ACTION Correction:
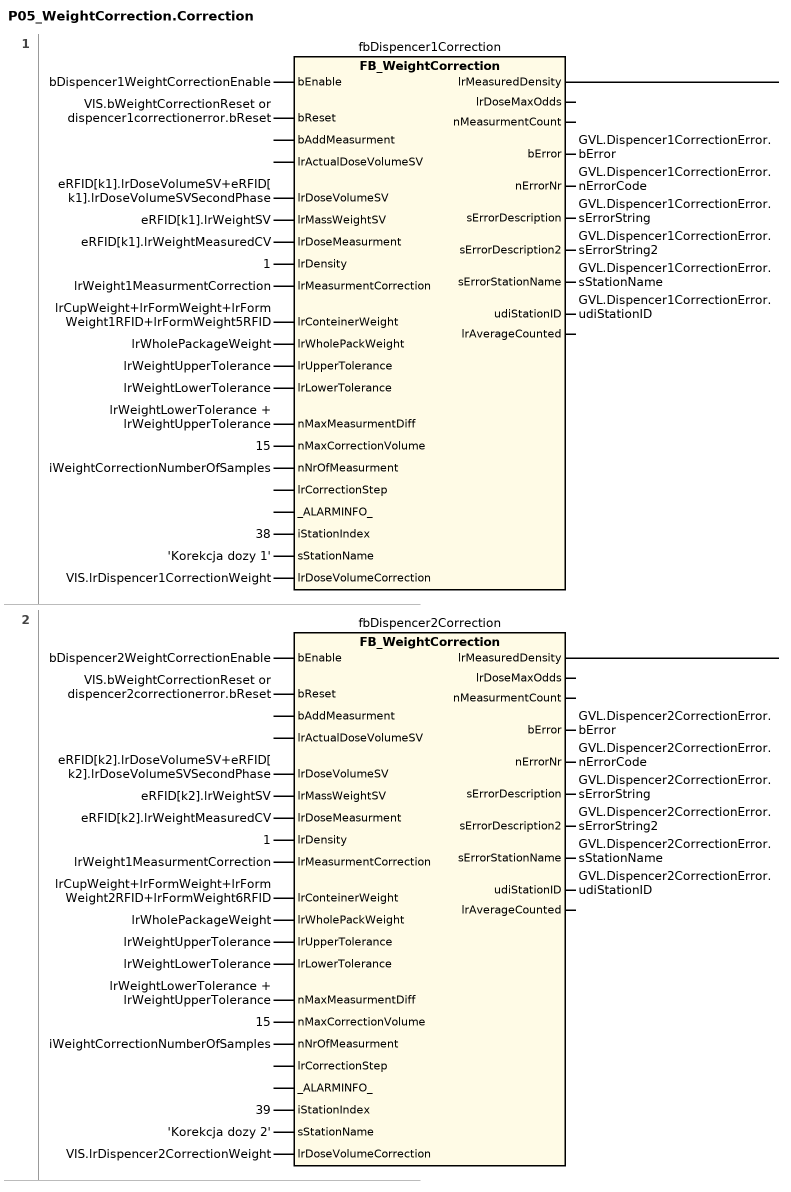
// NETWORK 1
fbDispencer1Correction(
    bEnable := bDispencer1WeightCorrectionEnable,
    bReset := VIS.bWeightCorrectionReset or dispencer1correctionerror.bReset,
    lrDoseVolumeSV := eRFID[k1].lrDoseVolumeSV+eRFID[k1].lrDoseVolumeSVSecondPhase,
    lrMassWeightSV := eRFID[k1].lrWeightSV,
    lrDoseMeasurment := eRFID[k1].lrWeightMeasuredCV,
    lrDensity := 1,
    lrMeasurmentCorrection := lrWeight1MeasurmentCorrection,
    lrConteinerWeight := lrCupWeight+lrFormWeight+lrFormWeight1RFID+lrFormWeight5RFID,
    lrWholePackWeight := lrWholePackageWeight,
    lrUpperTolerance := lrWeightUpperTolerance,
    lrLowerTolerance := lrWeightLowerTolerance,
    nMaxMeasurmentDiff := lrWeightLowerTolerance + lrWeightUpperTolerance,
    nMaxCorrectionVolume := 15,
    nNrOfMeasurment := iWeightCorrectionNumberOfSamples,
    iStationIndex := 38,
    sStationName := 'Korekcja dozy 1',
    lrDoseVolumeCorrection := VIS.lrDispencer1CorrectionWeight,
    bError => GVL.Dispencer1CorrectionError.bError,
    nErrorNr => GVL.Dispencer1CorrectionError.nErrorCode,
    sErrorDescription => GVL.Dispencer1CorrectionError.sErrorString,
    sErrorDescription2 => GVL.Dispencer1CorrectionError.sErrorString2,
    sErrorStationName => GVL.Dispencer1CorrectionError.sStationName,
    udiStationID => GVL.Dispencer1CorrectionError.udiStationID); // FB_WeightCorrection

// NETWORK 2
fbDispencer2Correction(
    bEnable := bDispencer2WeightCorrectionEnable,
    bReset := VIS.bWeightCorrectionReset or dispencer2correctionerror.bReset,
    lrDoseVolumeSV := eRFID[k2].lrDoseVolumeSV+eRFID[k2].lrDoseVolumeSVSecondPhase,
    lrMassWeightSV := eRFID[k2].lrWeightSV,
    lrDoseMeasurment := eRFID[k2].lrWeightMeasuredCV,
    lrDensity := 1,
    lrMeasurmentCorrection := lrWeight1MeasurmentCorrection,
    lrConteinerWeight := lrCupWeight+lrFormWeight+lrFormWeight2RFID+lrFormWeight6RFID,
    lrWholePackWeight := lrWholePackageWeight,
    lrUpperTolerance := lrWeightUpperTolerance,
    lrLowerTolerance := lrWeightLowerTolerance,
    nMaxMeasurmentDiff := lrWeightLowerTolerance + lrWeightUpperTolerance,
    nMaxCorrectionVolume := 15,
    nNrOfMeasurment := iWeightCorrectionNumberOfSamples,
    iStationIndex := 39,
    sStationName := 'Korekcja dozy 2',
    lrDoseVolumeCorrection := VIS.lrDispencer2CorrectionWeight,
    bError => GVL.Dispencer2CorrectionError.bError,
    nErrorNr => GVL.Dispencer2CorrectionError.nErrorCode,
    sErrorDescription => GVL.Dispencer2CorrectionError.sErrorString,
    sErrorDescription2 => GVL.Dispencer2CorrectionError.sErrorString2,
    sErrorStationName => GVL.Dispencer2CorrectionError.sStationName,
    udiStationID => GVL.Dispencer2CorrectionError.udiStationID); // FB_WeightCorrection

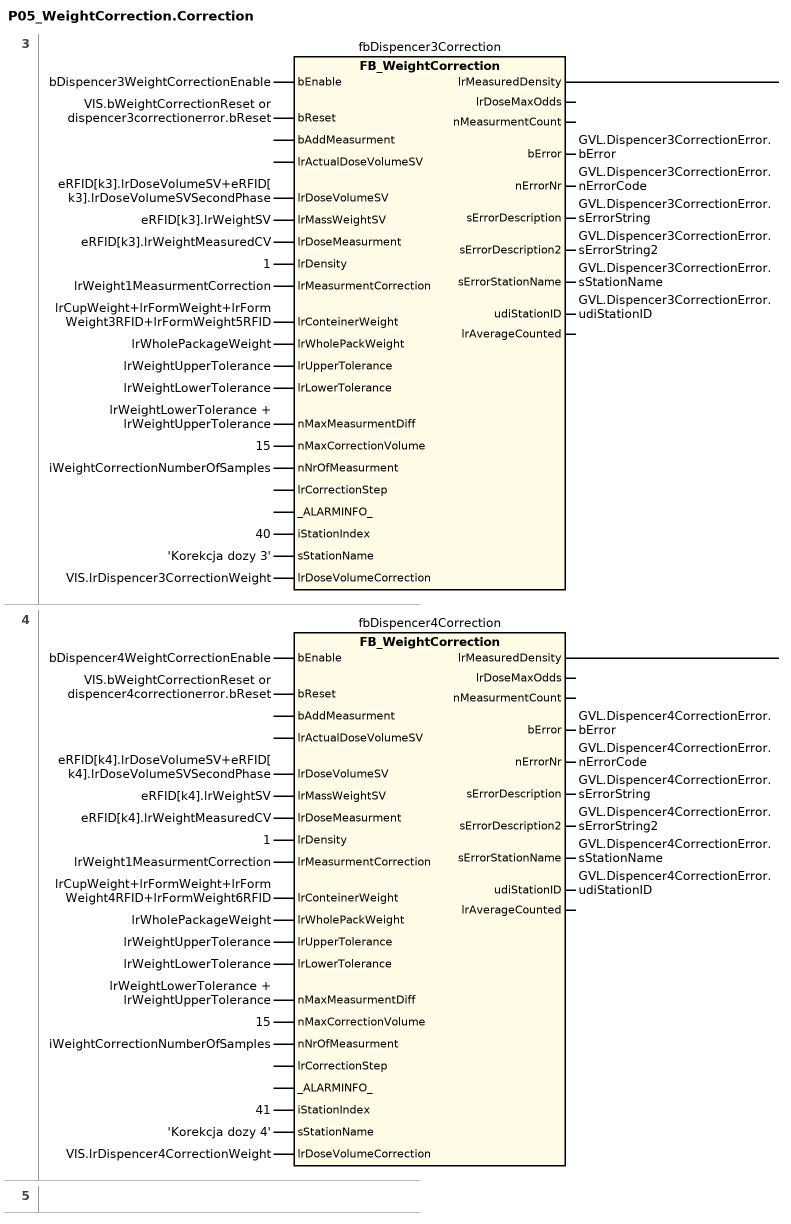
// NETWORK 3
fbDispencer3Correction(
    bEnable := bDispencer3WeightCorrectionEnable,
    bReset := VIS.bWeightCorrectionReset or dispencer3correctionerror.bReset,
    lrDoseVolumeSV := eRFID[k3].lrDoseVolumeSV+eRFID[k3].lrDoseVolumeSVSecondPhase,
    lrMassWeightSV := eRFID[k3].lrWeightSV,
    lrDoseMeasurment := eRFID[k3].lrWeightMeasuredCV,
    lrDensity := 1,
    lrMeasurmentCorrection := lrWeight1MeasurmentCorrection,
    lrConteinerWeight := lrCupWeight+lrFormWeight+lrFormWeight3RFID+lrFormWeight5RFID,
    lrWholePackWeight := lrWholePackageWeight,
    lrUpperTolerance := lrWeightUpperTolerance,
    lrLowerTolerance := lrWeightLowerTolerance,
    nMaxMeasurmentDiff := lrWeightLowerTolerance + lrWeightUpperTolerance,
    nMaxCorrectionVolume := 15,
    nNrOfMeasurment := iWeightCorrectionNumberOfSamples,
    iStationIndex := 40,
    sStationName := 'Korekcja dozy 3',
    lrDoseVolumeCorrection := VIS.lrDispencer3CorrectionWeight,
    bError => GVL.Dispencer3CorrectionError.bError,
    nErrorNr => GVL.Dispencer3CorrectionError.nErrorCode,
    sErrorDescription => GVL.Dispencer3CorrectionError.sErrorString,
    sErrorDescription2 => GVL.Dispencer3CorrectionError.sErrorString2,
    sErrorStationName => GVL.Dispencer3CorrectionError.sStationName,
    udiStationID => GVL.Dispencer3CorrectionError.udiStationID); // FB_WeightCorrection

// NETWORK 4
fbDispencer4Correction(
    bEnable := bDispencer4WeightCorrectionEnable,
    bReset := VIS.bWeightCorrectionReset or dispencer4correctionerror.bReset,
    lrDoseVolumeSV := eRFID[k4].lrDoseVolumeSV+eRFID[k4].lrDoseVolumeSVSecondPhase,
    lrMassWeightSV := eRFID[k4].lrWeightSV,
    lrDoseMeasurment := eRFID[k4].lrWeightMeasuredCV,
    lrDensity := 1,
    lrMeasurmentCorrection := lrWeight1MeasurmentCorrection,
    lrConteinerWeight := lrCupWeight+lrFormWeight+lrFormWeight4RFID+lrFormWeight6RFID,
    lrWholePackWeight := lrWholePackageWeight,
    lrUpperTolerance := lrWeightUpperTolerance,
    lrLowerTolerance := lrWeightLowerTolerance,
    nMaxMeasurmentDiff := lrWeightLowerTolerance + lrWeightUpperTolerance,
    nMaxCorrectionVolume := 15,
    nNrOfMeasurment := iWeightCorrectionNumberOfSamples,
    iStationIndex := 41,
    sStationName := 'Korekcja dozy 4',
    lrDoseVolumeCorrection := VIS.lrDispencer4CorrectionWeight,
    bError => GVL.Dispencer4CorrectionError.bError,
    nErrorNr => GVL.Dispencer4CorrectionError.nErrorCode,
    sErrorDescription => GVL.Dispencer4CorrectionError.sErrorString,
    sErrorDescription2 => GVL.Dispencer4CorrectionError.sErrorString2,
    sErrorStationName => GVL.Dispencer4CorrectionError.sStationName,
    udiStationID => GVL.Dispencer4CorrectionError.udiStationID); // FB_WeightCorrection

// NETWORK 5
END_ACTION

ACTION OnePhaseDosing:
	(*******Dozowanie jednofazowe*****)

IF rtWeightingDone.Q THEN //Triger, wszystko wazy się jednoczesnie
	
	FOR i := 1 TO 100 DO
		
		IF  eWeightPackageState[1].nCardNumber = eRFID[i].nCardNumber AND eRFID[i].nDispencerNr=1 THEN	 
			
			fbDispencer1Correction.bAddMeasurment:=(eRFID[i].nDispencerNr=1 AND bDispencer1WeightCorrectionEnable) AND 
								(eRFID[i].lrDoseVolumeCV>(0.5*eRFID[i].lrDoseVolumeSV) OR eRFID[i].lrDoseVolumeCVSecondPhase>(0.5*eRFID[i].lrDoseVolumeSVSecondPhase)) AND
								(eRFID[i].lrWeightMeasuredCV>0);															
			k1:=i;	//Zapamiętywanie numeru tablicy		
			
			IF 					(eRFID[i].nDispencerNr=1 AND bDispencer1WeightCorrectionEnable) AND 
								((eRFID[i].lrDoseVolumeCV>(0.5*eRFID[i].lrDoseVolumeSV)) OR (eRFID[i].lrDoseVolumeCVSecondPhase>(0.5*eRFID[i].lrDoseVolumeSVSecondPhase))) AND
								(eRFID[i].lrWeightMeasuredCV>0) THEN
				iCorectTest:=iCorectTest+1;	
			END_IF;	
		END_IF	
    
		IF  eWeightPackageState[1].nCardNumber = eRFID[i].nCardNumber AND eRFID[i].nDispencerNr=2 THEN	
 
			fbDispencer2Correction.bAddMeasurment := (eRFID[i].nDispencerNr=2 AND bDispencer2WeightCorrectionEnable) AND 
								(eRFID[i].lrDoseVolumeCV>(0.5*eRFID[i].lrDoseVolumeSV) OR eRFID[i].lrDoseVolumeCVSecondPhase>(0.5*eRFID[i].lrDoseVolumeSVSecondPhase)) AND 
								(eRFID[i].lrWeightMeasuredCV>0);
			k2:=i;	//Zapamiętywanie numeru tablicy	
			iCorectTest2:=iCorectTest2+1;							
		END_IF
		
		IF  eWeightPackageState[1].nCardNumber = eRFID[i].nCardNumber AND eRFID[i].nDispencerNr=3 THEN	 
			fbDispencer3Correction.bAddMeasurment := (eRFID[i].nDispencerNr=3 AND bDispencer3WeightCorrectionEnable) AND 
								(eRFID[i].lrDoseVolumeCV>(0.5*eRFID[i].lrDoseVolumeSV) OR eRFID[i].lrDoseVolumeCVSecondPhase>(0.5*eRFID[i].lrDoseVolumeSVSecondPhase)) AND 
								(eRFID[i].lrWeightMeasuredCV>0);						
			k3:=i;	//Zapamiętywanie numeru tablicy		
			iCorectTest3:=iCorectTest3+1;					
		END_IF	
		
		IF  eWeightPackageState[1].nCardNumber = eRFID[i].nCardNumber AND eRFID[i].nDispencerNr=4 THEN	 
			fbDispencer4Correction.bAddMeasurment := (eRFID[i].nDispencerNr=4 AND bDispencer4WeightCorrectionEnable) AND 
								(eRFID[i].lrDoseVolumeCV>(0.5*eRFID[i].lrDoseVolumeSV) OR eRFID[i].lrDoseVolumeCVSecondPhase>(0.5*eRFID[i].lrDoseVolumeSVSecondPhase)) AND 
								(eRFID[i].lrWeightMeasuredCV>0);					
			k4:=i;	//Zapamiętywanie numeru tablicy	
			iCorectTest4:=iCorectTest4+1;						
		END_IF
		
	END_FOR
	
	
	FOR i := 1 TO 100 DO
		
		IF  eWeightPackageState[2].nCardNumber = eRFID[i].nCardNumber AND eRFID[i].nDispencerNr=1 THEN	 
			fbDispencer1Correction.bAddMeasurment:=(eRFID[i].nDispencerNr=1 AND bDispencer1WeightCorrectionEnable) AND 
								(eRFID[i].lrDoseVolumeCV>(0.5*eRFID[i].lrDoseVolumeSV) OR eRFID[i].lrDoseVolumeCVSecondPhase>(0.5*eRFID[i].lrDoseVolumeSVSecondPhase)) AND
								(eRFID[i].lrWeightMeasuredCV>0);															
			k1:=i;	//Zapamiętywanie numeru tablicy						
		END_IF	
		
		IF  eWeightPackageState[2].nCardNumber = eRFID[i].nCardNumber AND eRFID[i].nDispencerNr=2 THEN	 
			fbDispencer2Correction.bAddMeasurment := (eRFID[i].nDispencerNr=2 AND bDispencer2WeightCorrectionEnable) AND 
								(eRFID[i].lrDoseVolumeCV>(0.5*eRFID[i].lrDoseVolumeSV) OR eRFID[i].lrDoseVolumeCVSecondPhase>(0.5*eRFID[i].lrDoseVolumeSVSecondPhase)) AND 
								(eRFID[i].lrWeightMeasuredCV>0);
			k2:=i;	//Zapamiętywanie numeru tablicy						
		END_IF
		
		IF  eWeightPackageState[2].nCardNumber = eRFID[i].nCardNumber AND eRFID[i].nDispencerNr=3 THEN	 
			fbDispencer3Correction.bAddMeasurment := (eRFID[i].nDispencerNr=3 AND bDispencer3WeightCorrectionEnable) AND 
								(eRFID[i].lrDoseVolumeCV>(0.5*eRFID[i].lrDoseVolumeSV) OR eRFID[i].lrDoseVolumeCVSecondPhase>(0.5*eRFID[i].lrDoseVolumeSVSecondPhase)) AND 
								(eRFID[i].lrWeightMeasuredCV>0);						
			k3:=i;	//Zapamiętywanie numeru tablicy						
		END_IF	
		
		IF  eWeightPackageState[2].nCardNumber = eRFID[i].nCardNumber AND eRFID[i].nDispencerNr=4 THEN	 
			fbDispencer4Correction.bAddMeasurment := (eRFID[i].nDispencerNr=4 AND bDispencer4WeightCorrectionEnable) AND 
								(eRFID[i].lrDoseVolumeCV>(0.5*eRFID[i].lrDoseVolumeSV) OR eRFID[i].lrDoseVolumeCVSecondPhase>(0.5*eRFID[i].lrDoseVolumeSVSecondPhase)) AND 
								(eRFID[i].lrWeightMeasuredCV>0);					
			k4:=i;	//Zapamiętywanie numeru tablicy						
		END_IF
		
	END_FOR		
    
	FOR i := 1 TO 100 DO
		
		IF  eWeightPackageState[3].nCardNumber = eRFID[i].nCardNumber  AND eRFID[i].nDispencerNr=1 THEN	 
			fbDispencer1Correction.bAddMeasurment:=(eRFID[i].nDispencerNr=1 AND bDispencer1WeightCorrectionEnable) AND 
								(eRFID[i].lrDoseVolumeCV>(0.5*eRFID[i].lrDoseVolumeSV) OR eRFID[i].lrDoseVolumeCVSecondPhase>(0.5*eRFID[i].lrDoseVolumeSVSecondPhase)) AND
								(eRFID[i].lrWeightMeasuredCV>0);															
			k1:=i;	//Zapamiętywanie numeru tablicy						
		END_IF	
		
		IF  eWeightPackageState[3].nCardNumber = eRFID[i].nCardNumber AND eRFID[i].nDispencerNr=2 THEN	 
			fbDispencer2Correction.bAddMeasurment := (eRFID[i].nDispencerNr=2 AND bDispencer2WeightCorrectionEnable) AND 
								(eRFID[i].lrDoseVolumeCV>(0.5*eRFID[i].lrDoseVolumeSV) OR eRFID[i].lrDoseVolumeCVSecondPhase>(0.5*eRFID[i].lrDoseVolumeSVSecondPhase)) AND 
								(eRFID[i].lrWeightMeasuredCV>0);
			k2:=i;	//Zapamiętywanie numeru tablicy						
		END_IF
		
		IF  eWeightPackageState[3].nCardNumber = eRFID[i].nCardNumber AND eRFID[i].nDispencerNr=3 THEN	 
			fbDispencer3Correction.bAddMeasurment := (eRFID[i].nDispencerNr=3 AND bDispencer3WeightCorrectionEnable) AND 
								(eRFID[i].lrDoseVolumeCV>(0.5*eRFID[i].lrDoseVolumeSV) OR eRFID[i].lrDoseVolumeCVSecondPhase>(0.5*eRFID[i].lrDoseVolumeSVSecondPhase)) AND 
								(eRFID[i].lrWeightMeasuredCV>0);						
			k3:=i;	//Zapamiętywanie numeru tablicy						
		END_IF	
		
		IF  eWeightPackageState[3].nCardNumber = eRFID[i].nCardNumber AND eRFID[i].nDispencerNr=4 THEN	 
			fbDispencer4Correction.bAddMeasurment := (eRFID[i].nDispencerNr=4 AND bDispencer4WeightCorrectionEnable) AND 
								(eRFID[i].lrDoseVolumeCV>(0.5*eRFID[i].lrDoseVolumeSV) OR eRFID[i].lrDoseVolumeCVSecondPhase>(0.5*eRFID[i].lrDoseVolumeSVSecondPhase)) AND 
								(eRFID[i].lrWeightMeasuredCV>0);					
			k4:=i;	//Zapamiętywanie numeru tablicy						
		END_IF
		
	END_FOR
    
	FOR i := 1 TO 100 DO
		
		IF  eWeightPackageState[4].nCardNumber = eRFID[i].nCardNumber AND eRFID[i].nDispencerNr=1 THEN	 
			fbDispencer1Correction.bAddMeasurment:=(eRFID[i].nDispencerNr=1 AND bDispencer1WeightCorrectionEnable) AND 
								(eRFID[i].lrDoseVolumeCV>(0.5*eRFID[i].lrDoseVolumeSV) OR eRFID[i].lrDoseVolumeCVSecondPhase>(0.5*eRFID[i].lrDoseVolumeSVSecondPhase)) AND
								(eRFID[i].lrWeightMeasuredCV>0);															
			k1:=i;	//Zapamiętywanie numeru tablicy						
		END_IF	
		
		IF  eWeightPackageState[4].nCardNumber = eRFID[i].nCardNumber AND eRFID[i].nDispencerNr=2 THEN	 
			fbDispencer2Correction.bAddMeasurment := (eRFID[i].nDispencerNr=2 AND bDispencer2WeightCorrectionEnable) AND 
								(eRFID[i].lrDoseVolumeCV>(0.5*eRFID[i].lrDoseVolumeSV) OR eRFID[i].lrDoseVolumeCVSecondPhase>(0.5*eRFID[i].lrDoseVolumeSVSecondPhase)) AND 
								(eRFID[i].lrWeightMeasuredCV>0);
			k2:=i;	//Zapamiętywanie numeru tablicy						
		END_IF
		
		IF  eWeightPackageState[4].nCardNumber = eRFID[i].nCardNumber AND eRFID[i].nDispencerNr=3 THEN	 
			fbDispencer3Correction.bAddMeasurment := (eRFID[i].nDispencerNr=3 AND bDispencer3WeightCorrectionEnable) AND 
								(eRFID[i].lrDoseVolumeCV>(0.5*eRFID[i].lrDoseVolumeSV) OR eRFID[i].lrDoseVolumeCVSecondPhase>(0.5*eRFID[i].lrDoseVolumeSVSecondPhase)) AND 
								(eRFID[i].lrWeightMeasuredCV>0);						
			k3:=i;	//Zapamiętywanie numeru tablicy						
		END_IF
	
		IF  eWeightPackageState[4].nCardNumber = eRFID[i].nCardNumber AND eRFID[i].nDispencerNr=4 THEN	 
			fbDispencer4Correction.bAddMeasurment := (eRFID[i].nDispencerNr=4 AND bDispencer4WeightCorrectionEnable) AND 
								(eRFID[i].lrDoseVolumeCV>(0.5*eRFID[i].lrDoseVolumeSV) OR eRFID[i].lrDoseVolumeCVSecondPhase>(0.5*eRFID[i].lrDoseVolumeSVSecondPhase)) AND 
								(eRFID[i].lrWeightMeasuredCV>0);					
			k4:=i;	//Zapamiętywanie numeru tablicy						
		END_IF
		
	END_FOR

END_IF
END_ACTION

ACTION TwoPhaseDosing:
	(*******Dozowanie jednofazowe*****)

IF rtWeightingDone.Q THEN //Triger, wszystko wazy się jednoczesnie
	
	FOR i2 := 1 TO 100 DO
		
		IF  eWeightPackage2PhasePackageState[1].nCardNumber = eRFID[i2].nCardNumber AND (*eRFID[i2].nDispencerNr=1*) eRFID[i2].nDispencerNrSecondPhase=1 THEN	 
			
			fbDispencer1Correction.bAddMeasurment:=((*eRFID[i2].nDispencerNr=1 AND*) eRFID[i2].nDispencerNrSecondPhase=1 AND bDispencer1WeightCorrectionEnable) AND 
								(eRFID[i2].lrDoseVolumeCV>(0.5*eRFID[i2].lrDoseVolumeSV) OR eRFID[i2].lrDoseVolumeCVSecondPhase>(0.5*eRFID[i2].lrDoseVolumeSVSecondPhase)) AND
								(eRFID[i2].lrWeightMeasuredCV>0);															
			k1:=i2;	//Zapamiętywanie numeru tablicy		
			iCorectTest:=iCorectTest+1;
		END_IF	
	END_FOR
	
	FOR i3:=1 TO 100 DO
	
    (*
		IF  eWeightPackage2PhasePackageState[1].nCardNumber = eRFID[i2].nCardNumber AND (*eRFID[i2].nDispencerNr=2*) eRFID[i2].nDispencerNrSecondPhase=2 THEN	
 
			fbDispencer2Correction.bAddMeasurment := ((*eRFID[i2].nDispencerNr=2*)eRFID[i2].nDispencerNrSecondPhase=2 AND bDispencer2WeightCorrectionEnable) AND 
								(eRFID[i2].lrDoseVolumeCV>(0.5*eRFID[i2].lrDoseVolumeSV) OR eRFID[i2].lrDoseVolumeCVSecondPhase>(0.5*eRFID[i2].lrDoseVolumeSVSecondPhase)) AND 
								(eRFID[i2].lrWeightMeasuredCV>0);
			k2:=i2;	//Zapamiętywanie numeru tablicy	
			iCorectTest2:=iCorectTest2+1;	
			EXIT;						
		END_IF
	*)	
		IF  eWeightPackage2PhasePackageState[1].nCardNumber = eRFID[i3].nCardNumber AND eRFID[i3].nDispencerNr=3 THEN	 
			fbDispencer3Correction.bAddMeasurment := (eRFID[i3].nDispencerNr=3 AND bDispencer3WeightCorrectionEnable) AND 
								(eRFID[i3].lrDoseVolumeCV>(0.5*eRFID[i3].lrDoseVolumeSV) OR eRFID[i3].lrDoseVolumeCVSecondPhase>(0.5*eRFID[i3].lrDoseVolumeSVSecondPhase)) AND 
								(eRFID[i3].lrWeightMeasuredCV>0);						
			k3:=i3;	//Zapamiętywanie numeru tablicy		
			iCorectTest3:=iCorectTest3+1;	
						
		END_IF	
	(*	
		IF  eWeightPackage2PhasePackageState[1].nCardNumber = eRFID[i2].nCardNumber AND eRFID[i2].nDispencerNr=4 THEN	 
			fbDispencer4Correction.bAddMeasurment := (eRFID[i2].nDispencerNr=4 AND bDispencer4WeightCorrectionEnable) AND 
								(eRFID[i2].lrDoseVolumeCV>(0.5*eRFID[i2].lrDoseVolumeSV) OR eRFID[i2].lrDoseVolumeCVSecondPhase>(0.5*eRFID[i2].lrDoseVolumeSVSecondPhase)) AND 
								(eRFID[i2].lrWeightMeasuredCV>0);					
			k4:=i2;	//Zapamiętywanie numeru tablicy	
			iCorectTest4:=iCorectTest4+1;	
			EXIT;					
		END_IF
	*)	

	END_FOR
	
	
	FOR i4 := 1 TO 100 DO
		(*
		IF  eWeightPackage2PhasePackageState[2].nCardNumber = eRFID[i].nCardNumber AND eRFID[i].nDispencerNr=1 THEN	 
			fbDispencer1Correction.bAddMeasurment:=(eRFID[i].nDispencerNr=1 AND bDispencer1WeightCorrectionEnable) AND 
								(eRFID[i].lrDoseVolumeCV>(0.5*eRFID[i].lrDoseVolumeSV) OR eRFID[i].lrDoseVolumeCVSecondPhase>(0.5*eRFID[i].lrDoseVolumeSVSecondPhase)) AND
								(eRFID[i].lrWeightMeasuredCV>0);															
			k1:=i;	//Zapamiętywanie numeru tablicy	
			iCorectTest5:=iCorectTest5+1;	
		EXIT;			
		END_IF	
		*)
		IF  eWeightPackage2PhasePackageState[2].nCardNumber = eRFID[i4].nCardNumber AND (*eRFID[i].nDispencerNr=2*) eRFID[i4].nDispencerNrSecondPhase=2 THEN	 
			fbDispencer2Correction.bAddMeasurment := ((*eRFID[i].nDispencerNr=2*) eRFID[i4].nDispencerNrSecondPhase=2 AND bDispencer2WeightCorrectionEnable) AND 
								(eRFID[i4].lrDoseVolumeCV>(0.5*eRFID[i4].lrDoseVolumeSV) OR eRFID[i4].lrDoseVolumeCVSecondPhase>(0.5*eRFID[i4].lrDoseVolumeSVSecondPhase)) AND 
								(eRFID[i4].lrWeightMeasuredCV>0);
			k2:=i4;	//Zapamiętywanie numeru tablicy		
			iCorectTest6:=iCorectTest6+1;	
		END_IF
	END_FOR
	
	FOR i5:=1 TO 100 DO
		(*
		IF  eWeightPackage2PhasePackageState[2].nCardNumber = eRFID[i].nCardNumber AND eRFID[i].nDispencerNr=3 THEN	 
			fbDispencer3Correction.bAddMeasurment := (eRFID[i].nDispencerNr=3 AND bDispencer3WeightCorrectionEnable) AND 
								(eRFID[i].lrDoseVolumeCV>(0.5*eRFID[i].lrDoseVolumeSV) OR eRFID[i].lrDoseVolumeCVSecondPhase>(0.5*eRFID[i].lrDoseVolumeSVSecondPhase)) AND 
								(eRFID[i].lrWeightMeasuredCV>0);						
			k3:=i;	//Zapamiętywanie numeru tablicy	
			iCorectTest7:=iCorectTest7+1;	
		EXIT	;			
		END_IF	
		*)
		IF  eWeightPackage2PhasePackageState[2].nCardNumber = eRFID[i5].nCardNumber AND eRFID[i5].nDispencerNr=4  THEN	 
			fbDispencer4Correction.bAddMeasurment := (eRFID[i5].nDispencerNr=4 AND bDispencer4WeightCorrectionEnable) AND 
								(eRFID[i5].lrDoseVolumeCV>(0.5*eRFID[i5].lrDoseVolumeSV) OR eRFID[i5].lrDoseVolumeCVSecondPhase>(0.5*eRFID[i5].lrDoseVolumeSVSecondPhase)) AND 
								(eRFID[i5].lrWeightMeasuredCV>0);					
			k4:=i5;	//Zapamiętywanie numeru tablicy	
			iCorectTest8:=iCorectTest8+1;	
		END_IF
		
	END_FOR		
    


END_IF
END_ACTION

END_PROGRAM

// ---- POUs/FB/FB_WeightCorrection.TcPOU
(*
Nazwa:			FB_WeightCorrection
Opis:			Korekcja wagi
Wersja:			v1.3
Data:			2019-11-28
Autor:			TW,DP
Urzadzenia:		Korekta wagi 
Konfiguracja:	
Info: 
-wyłączono wpisywanie maksymalnej korekty bo to bez sensu, ze wpisywało np -15
-poprawiono warningi, które wskazywalo w kompilatorze
-poprawiony blad maksymalnej korekty (minus przerabia na plus)
*)

FUNCTION_BLOCK FB_WeightCorrection
VAR_INPUT
	bEnable:BOOL;					//Zezwolenie na pracę automatycznej korekcji
	bReset:BOOL;					//Reset korekcji dozy i obliczonej gęstości
	bAddMeasurment:BOOL;			//Dodanie pomiaru wagi do rozpatrzenia korekcji dozy
	lrActualDoseVolumeSV:LREAL;		//Aktualna wartość nastawy objetości dozy (ta która jest nastawiona na dozowniku)
	lrDoseVolumeSV:LREAL;			//Wartość nastawy objetości dozy dla danego opakowania (wartość z rejestru)  [ml]
	lrMassWeightSV:LREAL;			//Zadana wartość masy produktu [g]
	lrDoseMeasurment:LREAL;			//Wartość masy odczytana z wagi [g]
	lrDensity:LREAL;				//Gęstość masy g/ml (Jeśli wartość 0, oblicz z wydozowanej ostatniej wartości)
	lrMeasurmentCorrection:LREAL;	//Korekcja wskazania wagi [g]
	lrConteinerWeight:LREAL;			//Waga kubeczka [g]
	lrWholePackWeight:LREAL;		//Waga kubeczka razem z platynką i nakrętką itp. [g]
	lrUpperTolerance:LREAL;			//Górna granica tolerancji
	lrLowerTolerance:LREAL;			//Dolna granica tolerancji	
	nMaxMeasurmentDiff:LREAL;		//Maksymalna różnica pomiędzy pomiarami
	nMaxCorrectionVolume:UDINT;		//Maksymalna nastawa dozy korekcji
	nNrOfMeasurment:UINT;			//Ilość próbek do uśrednienia wartości korekcji dozy
	lrCorrectionStep: LREAL;		//Skok korekcji dozy [ml]
	_ALARMINFO_ :BOOL;
	iStationIndex:UDINT;					//Numer stacji 
	sStationName:STRING;					//Nazwa stacji	

END_VAR
VAR_OUTPUT
	lrMeasuredDensity:LREAL;		//Obliczona wartość gęstości [g/ml]
	lrDoseMaxOdds:LREAL;			//Najwieksze różnice pomiędzy wagami wydozowań
	nMeasurmentCount:UINT;			//Ilość zebranych pomiarów do uśrednienia wagi
	bError:BOOL; 					//Błąd korekcji <=0
	nErrorNr:UDINT;					//Numer Błędu
	sErrorDescription:STRING;		//Opis błędu 
	sErrorDescription2: STRING;				//Opis błędu 2
	sErrorStationName:STRING;				//Nazwa stacji
	udiStationID:UDINT;				// Nr stacji

	lrAverageCounted:LREAL;			//średnia z ostatnich pomiarów
END_VAR
VAR_IN_OUT
	lrDoseVolumeCorrection:LREAL;			//Wartość korekty dozy [ml]
END_VAR
VAR
	rtAddMeasurment: R_TRIG;
	aMeasuredWeight: ARRAY [1..10] OF LREAL;
	
	i: UINT;
	// Suma pomiarów wag
	lrMeasureSum: LREAL;
	// Średnia pomiarów wagi
	lrAverageWeight: LREAL;
	lrUsedDensity:LREAL;
	// trigger Resetu
	rtrigReset: R_TRIG;
	// poprzednia wartość dozy kontrolowanej butelki [ml]
	lrLastDoseVolumeSV: LREAL :=89033008911;
	lrDoseVolumeCorrectionTemp: LREAL;
	Delta: DINT;
	bWeightTooLow:BOOL;
	bWeightTooHigh:BOOL;
	lrWeightHisteresisCenter:LREAL;//
END_VAR

aStationID();
rtAddMeasurment(CLK:=bAddMeasurment,Q=>);


IF bEnable THEN
	
	
	//Jeśli odczytana nowa doza 
	IF rtAddMeasurment.Q THEN
		
		//Jeśli dozy różne zacznij próbkowanie wag od początku
		IF lrActualDoseVolumeSV<>lrDoseVolumeSV THEN
			nMeasurmentCount:=0;
			lrMeasureSum:=0;
		
		//jeśli nastawy zgadzają sie 	
		ELSE	
		
			lrLastDoseVolumeSV:=lrDoseVolumeSV;
			bError:=FALSE;
			nMeasurmentCount:=nMeasurmentCount+1;
			aMeasuredWeight[nMeasurmentCount]:=lrDoseMeasurment-lrConteinerWeight+lrMeasurmentCorrection;
			lrMeasureSum:=lrMeasureSum+aMeasuredWeight[nMeasurmentCount];
			
			IF nMeasurmentCount=1 THEN
				lrDoseMaxOdds:=0;
			END_IF
			
			//Sprawdzanie największych odchyłek w wadze miedzy pomiarami
			FOR i:=1 TO nMeasurmentCount DO
				IF ABS(aMeasuredWeight[i]-aMeasuredWeight[nMeasurmentCount])>lrDoseMaxOdds THEN
					lrDoseMaxOdds:=ABS(aMeasuredWeight[i]-aMeasuredWeight[nMeasurmentCount]);
				END_IF
			END_FOR
			

		END_IF
		
		IF lrDoseMaxOdds>nMaxMeasurmentDiff THEN
				nMeasurmentCount:=0;
				lrMeasureSum:=0;
		END_IF
		//Obliczanie korekty jeśli ilość próbek pomiarowych została osiągnięta
		IF nMeasurmentCount>=(nNrOfMeasurment) THEN
			lrAverageWeight:=lrMeasureSum/UINT_TO_LREAL(nMeasurmentCount);
			lrAverageCounted:=lrAverageWeight;
			lrMeasureSum:=0;
			//lrMeasuredDensity:=(lrAverageWeight)/(lrDoseVolumeSV(*+lrDoseVolumeCorrection*)+0.000000000001);
			IF lrDensity>0 THEN
				lrUsedDensity:=lrDensity;
			ELSE
				//lrUsedDensity:=lrMeasuredDensity;
				bError:=TRUE;
				nErrorNr:=211;
				sErrorDescription:='Zadana wartość gęstości poniżej 0.';
			END_IF
			
			
			//Jeśli nie ma błędu oblicz korektę
			IF NOT bError (*AND (((LREAL_TO_DINT(lrMassWeightSV)-LREAL_TO_DINT(lrAverageWeight))>=ABS(lrLowerTolerance)) OR (((LREAL_TO_DINT(lrAverageWeight)-LREAL_TO_DINT(lrMassWeightSV)>=ABS(lrUpperTolerance)))))*) THEN
				
			
				Delta:=(LREAL_TO_DINT(lrMassWeightSV)-LREAL_TO_DINT(lrAverageCounted));
				
			//	lrWeightHisteresisCenter:=(LREAL_TO_DINT(lrMassWeightSV)+((ABS(lrLowerTolerance)+ABS(lrUpperTolerance))/2)-(ABS(lrLowerTolerance)));
				// 04.11.2022 Dązy do zadanej bez środka
				lrWeightHisteresisCenter:=lrMassWeightSV;
				
				//Wykrywanie czy waga przekracza górny zakres widełek
				IF LREAL_TO_DINT(lrAverageCounted)<LREAL_TO_DINT(lrWeightHisteresisCenter) THEN
					bWeightTooLow:=TRUE;
					bWeightTooHigh:=FALSE;
			   //Wykrywanie czy waga przekracza dolną granicę widełek
				ELSIF LREAL_TO_DINT(lrAverageCounted)>LREAL_TO_DINT(lrWeightHisteresisCenter)THEN
					bWeightTooLow:=FALSE;
					bWeightTooHigh:=TRUE;
				END_IF
				
				
				
				//Jeśli osiągnieta wartość miedzy widełkami wyłącz podnoszenie dozy
				IF LREAL_TO_DINT(lrAverageCounted)>=(LREAL_TO_DINT(lrMassWeightSV)+((ABS(lrLowerTolerance)+ABS(lrUpperTolerance))/2)-(ABS(lrLowerTolerance))) THEN
					bWeightTooLow:=FALSE;
				END_IF
				
				//Jeśli osiągnieta wartość miedzy widełkami wyłącz obniżanie dozy
				IF LREAL_TO_DINT(lrAverageCounted)<=(LREAL_TO_DINT(lrMassWeightSV)+((ABS(lrLowerTolerance)+ABS(lrUpperTolerance))/2)-(ABS(lrLowerTolerance)))THEN
					bWeightTooHigh:=FALSE;
				END_IF
				
				//Zwiększ dozę jeśli za mała wartość
				IF bWeightTooLow THEN
					IF ABS(LREAL_TO_DINT(lrMassWeightSV)-LREAL_TO_DINT(lrAverageCounted))>10 THEN
						;//lrDoseVolumeCorrection:=lrDoseVolumeCorrection+ABS(LREAL_TO_DINT(lrMassWeightSV)-LREAL_TO_DINT(lrAverageCounted));//wyłączone max
					ELSE
						lrDoseVolumeCorrection:=lrDoseVolumeCorrection+lrCorrectionStep;	
					END_IF
						
						lrLastDoseVolumeSV:=lrDoseVolumeSV;
						
				//Zmniejsz dozę jeśli za duża	
				ELSIF bWeightTooHigh THEN
					IF ABS(LREAL_TO_DINT(lrMassWeightSV)-LREAL_TO_DINT(lrAverageCounted))>10 THEN
						;//lrDoseVolumeCorrection:=lrDoseVolumeCorrection-ABS(LREAL_TO_DINT(lrMassWeightSV)-LREAL_TO_DINT(lrAverageCounted));
					ELSE
						lrDoseVolumeCorrection:=lrDoseVolumeCorrection-lrCorrectionStep;	
					END_IF
					
					lrLastDoseVolumeSV:=lrDoseVolumeSV;
				END_IF
				
				//jeśli korekta poza maksymalnym zakresem, przepisz maksymalny zakres
				IF lrDoseVolumeCorrection>nMaxCorrectionVolume THEN					
					lrDoseVolumeCorrection:=nMaxCorrectionVolume;	
				END_IF
				IF lrDoseVolumeCorrection<-UDINT_TO_LREAL(nMaxCorrectionVolume) THEN					
					lrDoseVolumeCorrection:=-UDINT_TO_LREAL(nMaxCorrectionVolume);	
				END_IF
				
			END_IF;
			nMeasurmentCount:=0;
			lrAverageWeight:=0;
		END_IF	
	END_IF

ELSE
	nMeasurmentCount:=0;
	bError:=FALSE;
	lrDoseMaxOdds:=0;
END_IF

rtrigReset(CLK:=bReset,Q=>);

IF rtrigReset.Q (*AND NOT bError *)THEN
	nMeasurmentCount:=0;
	bError:=FALSE;
	lrDoseMaxOdds:=0;
	lrDoseVolumeCorrection:=0;
	lrMeasuredDensity:=0;
	lrMeasureSum:=0;
END_IF

ErrorHandling();

ACTION aStationID:
udiStationID	:=	iStationIndex;
END_ACTION

ACTION ErrorHandling:

IF bReset THEN
	bError:=FALSE;
	nErrorNr:=0;
	sErrorDescription:='';
	lrDoseMaxOdds:=0;
	lrDoseVolumeCorrectionTemp:=0;
END_IF

IF bEnable THEN
	;
	
ELSE
	bError:=FALSE;
	nErrorNr:=0;
	sErrorDescription:='';	
END_IF


(*Przepisywanie nazwy stacji*)
sErrorStationName := sStationName;
END_ACTION

END_FUNCTION_BLOCK

// ---- POUs/Recipes/P010_AlarmsWarningsInfosLogs.TcPOU
PROGRAM P010_AlarmsWarningsInfosLogs
VAR CONSTANT 
	iNumberOfStations									:	DINT:=46;	
	iMaxNumberOfErrors									:	DINT:=100;	
	iStartLinePositionY									:	INT:=0;		
	iLinePositionYStep									:	INT:=55;
	iNumberOfWarnings									:	INT:=13;
END_VAR

VAR	
	bWarning				:	BOOL;	
	bHistoryShowScreeen		:BOOL;
	//Wiska
	udiInfoCounter			:	UDINT;
	sInfoBitmapId			:	STRING	:=	'MainImages.InfoOff'	;
	udiInfoTxtColor 		:	UDINT	:=	16#FFFFFFFF;

	udiWarningCounter		:	UDINT;
	sWarningBitmapId		:	STRING	:=	'MainImages.WarningOff'	;
	udiWarningTxtColor 		:	UDINT	:=	16#FFFFFFFF;


	iAlarmCounter			:	DINT;
	sAlarmBitmapId			:	STRING	:=	'MainImages.ErrorOff'	;
	udiAlarmTxtColor 		:	UDINT	:=	16#FFFFFFFF;
	//

	aiLinePositionYErrors										:	ARRAY [0..iNumberOfStations] OF INT;
	iLinePositionXErrors										:	INT	:=	50;
	iStationInErrorCounter											:	INT;					
	
	aiLinePositionYWarnings										:	ARRAY [0..iNumberOfWarnings - 1] OF INT;
	iLinePositionXWarnings										:	INT	:=	50;
	iStationInWarningCounter									:	INT;
	iPrevStationInWarningCounter								:	INT:=-1;
				
	//stError												: 	ARRAY[0..iMaxNumberOfErrors] OF ST_Error;
	aActualErrorsArray									:	ARRAY[0..2,0..iMaxNumberOfErrors] OF WSTRING(120);//iNumberOfWarnings - 1
	//stWarning											: 	ARRAY[0..iNumberOfWarnings - 1] OF ST_Warning;
	aActualWarningsArray								:	ARRAY[0..1,0..19] OF WSTRING(120);//iNumberOfWarnings - 1
	
	i													:	DINT;
	k													:	INT;
	j													:	INT;
	
	diId												:	DINT	:=	-1;
	iPrevStationInErrorCounter							:	DINT	:=	-1;

	udiResetCase										:	UDINT;
	artReset											:	ARRAY [0..iMaxNumberOfErrors] OF R_TRIG;
	abReset												:	ARRAY [0.. iMaxNumberOfErrors] OF BOOL;
	udiWarningResetCase									:	UDINT;

	bInit												:	BOOL;
	
	diSelectedLine										:	DINT:= 1;
	diPrevSelectedLine									:	DINT:= -1;
	bShowErrorDescription								:	BOOL;
	
	iUnreadInfoRecordsCounter							:	INT:=0;					
	iPrevUnreadInfoRecordsCounter						:	INT:=-1;	

	rtPowerOn											:	R_TRIG;
	rtHomingDone										:	R_TRIG;
	rtSafetyReset										:	R_TRIG;
	rtSafetyInSafe										:	R_TRIG;
	rtAutomatStart										:	R_TRIG;
	rtAutomatStop										:	R_TRIG;
	
	tonStart											:	ton;
	
	aInfoRecords										:	ARRAY [0..1,0..255] OF WSTRING(120);
	iSelectedArrayIndex									:	INT;
		

	wsTemp												:	WSTRING(120);
	arhHistoricalError									:	ARRAY [0..iMaxNumberOfErrors] OF R_TRIG;
	arhHistoricalWarning								:	ARRAY [0..iNumberOfWarnings-1] OF R_TRIG;
	
	bStartedinAutomat									:	bool;
	fbMain												: 	INT;
	aHistoricalLogFiltered								:	ARRAY [0..2,0..2000] OF WSTRING(120);
	bErrorsShow											:	BOOL;						
	bWarningsShow										:	BOOL;						
	bInfosShow											:	BOOL;						
	bTest: BOOL;
END_VAR

VAR PERSISTENT
	aHistoricalLog										:	ARRAY [0..2,0..2000] OF WSTRING(120);
END_VAR


//ACT_HistoricalLog();
IF bTest THEN
	METH_FilterHistoryTable();
	bTest := FALSE;
END_IF

IF bHistoryShowScreeen THEN
	bInfosShow := NOT bInfosShow;
	METH_FilterHistoryTable();
END_IF

METHOD METH_AddHistoryRecord : BOOL
VAR_INPUT
	wsType	:	WSTRING;
	wsInfo	:	WSTRING(120);
END_VAR
FOR j:=1999 TO 1 BY -1 DO
	aHistoricalLog[0,j]										:= 	aHistoricalLog[0,j-1];
	aHistoricalLog[1,j]										:= 	aHistoricalLog[1,j-1];	
	aHistoricalLog[2,j]										:= 	aHistoricalLog[2,j-1];		
	
END_FOR
aHistoricalLog[0,0]											:= 	P020_RtcEffectivityOEE.wsActualDt;
aHistoricalLog[1,0]											:= 	wsType;	
aHistoricalLog[2,0]											:= 	wsInfo;	

P009_ReadSavePersistent.ACT_SaveRequest();
END_METHOD

METHOD METH_FilterHistoryTable : BOOL
VAR_INPUT
END_VAR
i:= 0;
FOR j:=0 TO 1999 DO
		aHistoricalLogFiltered[0,j]										:= 	"";
		aHistoricalLogFiltered[1,j]										:= 	"";	
		aHistoricalLogFiltered[2,j]										:= 	"";
	IF 	(bErrorsShow AND aHistoricalLog[1,j] = "Błąd") OR
		(bWarningsShow AND aHistoricalLog[1,j] = "Ostrz.") OR
		(bInfosShow AND aHistoricalLog[1,j] = "Info")
 	THEN
		aHistoricalLogFiltered[0,i]										:= 	aHistoricalLog[0,j];
		aHistoricalLogFiltered[1,i]										:= 	aHistoricalLog[1,j];	
		aHistoricalLogFiltered[2,i]										:= 	aHistoricalLog[2,j];			
		i := i + 1;	
	END_IF
END_FOR
END_METHOD

END_PROGRAM

// ---- POUs/Recipes/P020_RtcEffectivityOEE.TcPOU
PROGRAM P020_RtcEffectivityOEE
VAR
	//Wizka
	udiTotalCounter										:	UDINT;
	udiTotalefficiency									:	UDINT;

	//Rtc
	fbGetTime											:	NT_GetTime;				//FB getter RTC value
	tonDelay											:	TON;					//TON for delay between FB reading
	iCaseRtc											:	INT;					//Rtc case variable
	stActualTime										:	TIMESTRUCT;	

	wsActualDt											:	WSTRING := "00.00.0000 00:00:00";			
END_VAR

ACT_GetRtc();

ACTION ACT_GetRtc:
fbGetTime();
tonDelay(IN:=(iCaseRtc=2),PT:=T#200MS);
CASE iCaseRtc OF
	0:	//Start FB
		fbGetTime.START									:=	TRUE;
		iCaseRtc										:=	1;
	1:	//Wait #bysy signal
		IF (NOT fbGetTime.BUSY) THEN
			stActualTime								:=	fbGetTime.TIMESTR;
			fbGetTime.START								:=	FALSE;
			iCaseRtc									:=	2;
		END_IF
	2:	//Delay beetween reading RTC (for saving CPU time :) )
		IF (tonDelay.Q) THEN
			iCaseRtc									:=	0;
			wsActualDt:=METH_DateTimeArray_To_Wstring();
		END_IF
END_CASE
END_ACTION

METHOD METH_DateTimeArray_To_Wstring : WSTRING
VAR_INPUT
END_VAR
VAR 
	wsTmp												:	WSTRING;
END_VAR
IF (stActualTime.wDay<10) THEN
	wsTmp:="0";
END_IF
wsTmp:=WCONCAT(wsTmp,WCONCAT(UINT_TO_WSTRING(stActualTime.wDay),"."));

IF (stActualTime.wMonth<10) THEN
	wsTmp:=WCONCAT(wsTmp,"0");
END_IF
wsTmp:=WCONCAT(wsTmp,WCONCAT(UINT_TO_WSTRING(stActualTime.wMonth),"."));

IF (stActualTime.wYear<1000) THEN
	wsTmp:=WCONCAT(wsTmp,"0");
ELSIF (stActualTime.wYear<100) THEN
	wsTmp:=WCONCAT(wsTmp,"00");
ELSIF (stActualTime.wYear<10) THEN
	wsTmp:=WCONCAT(wsTmp,"000");
END_IF
wsTmp:=WCONCAT(wsTmp,WCONCAT(UINT_TO_WSTRING(stActualTime.wYear)," "));

IF (stActualTime.wHour<10) THEN
	wsTmp:=WCONCAT(wsTmp,"0");
END_IF
wsTmp:=WCONCAT(wsTmp,WCONCAT(UINT_TO_WSTRING(stActualTime.wHour),":"));
IF (stActualTime.wMinute<10) THEN
	wsTmp:=WCONCAT(wsTmp,"0");
END_IF
wsTmp:=WCONCAT(wsTmp,WCONCAT(UINT_TO_WSTRING(stActualTime.wMinute),":"));
IF (stActualTime.wSecond<10) THEN
	wsTmp:=WCONCAT(wsTmp,"0");
END_IF
wsTmp:=WCONCAT(wsTmp,UINT_TO_WSTRING(stActualTime.wSecond));
METH_DateTimeArray_To_Wstring:=wsTmp;
END_METHOD

END_PROGRAM

// ---- POUs/Recipes/P009_ReadSavePersistent.TcPOU
PROGRAM P009_ReadSavePersistent
VAR
	fbSave						:	FB_WritePersistentData;
	udiWriteCycle				:	UDINT;	
END_VAR

CASE (udiWriteCycle) OF
	0:
		;
	10:
		fbSave.START									:=	TRUE;
		udiWriteCycle									:=	20;
	20:
		IF (NOT fbSave.BUSY OR fbSave.ERR) THEN
			fbSave.START								:=	FALSE;
			udiWriteCycle								:=	0;	
		END_IF
END_CASE

fbSave.PORT												:=	851;
fbSave.TMOUT											:=	T#1000MS;

fbSave();

ACTION ACT_SaveRequest:
IF (udiWriteCycle = 0) THEN
	udiWriteCycle										:=	10;
END_IF
END_ACTION

END_PROGRAM

// ---- POUs/P_AdsLicenseServer.TcPOU
PROGRAM P_AdsLicenseServer
VAR
    fbWriteInd  : ADSWRITEIND;
    fbWriteRes  : ADSWRITERES;

    fbReadInd   : ADSREADIND;
    fbReadRes   : ADSREADRES;

    bClearWrite : BOOL := FALSE;
    bClearRead  : BOOL := FALSE;

    pWriteData  : POINTER TO STRING(80);
    sProductId  : STRING(80);

    sTrialToken : STRING(256) := 'NO_LICENSE';

    cIG_RequestTrial  : UDINT := 16#80000001; // must have MSB = 1
    cIG_GetTrialToken : UDINT := 16#80000002;
END_VAR

// --- HANDLE WRITE (request) ---
fbWriteInd(CLEAR := bClearWrite);
bClearWrite := FALSE;

IF fbWriteInd.VALID THEN
    IF fbWriteInd.IDXGRP = cIG_RequestTrial THEN
        pWriteData := fbWriteInd.DATAADDR;
        sProductId := pWriteData^; // assume it's null-terminated STRING

        sTrialToken := CONCAT('TRIAL_', sProductId); 
        sTrialToken := CONCAT(sTrialToken, '_OK');

        fbWriteRes(
            NETID    := fbWriteInd.NETID,
            PORT     := fbWriteInd.PORT,
            INVOKEID := fbWriteInd.INVOKEID,
            RESULT   := 0,
            RESPOND  := TRUE
        );
    ELSE
        fbWriteRes(
            NETID    := fbWriteInd.NETID,
            PORT     := fbWriteInd.PORT,
            INVOKEID := fbWriteInd.INVOKEID,
            RESULT   := 16#701,
            RESPOND  := TRUE
        );
    END_IF
    bClearWrite := TRUE;
END_IF

// --- HANDLE READ (client wants token) ---
fbReadInd(CLEAR := bClearRead);
bClearRead := FALSE;

IF fbReadInd.VALID THEN
    IF fbReadInd.IDXGRP = cIG_GetTrialToken THEN
        fbReadRes(
            NETID    := fbReadInd.NETID,
            PORT     := fbReadInd.PORT,
            INVOKEID := fbReadInd.INVOKEID,
            RESULT   := 0,
            LEN      := SIZEOF(sTrialToken),
            DATAADDR := ADR(sTrialToken),
            RESPOND  := TRUE
        );
    ELSE
        fbReadRes(
            NETID    := fbReadInd.NETID,
            PORT     := fbReadInd.PORT,
            INVOKEID := fbReadInd.INVOKEID,
            RESULT   := 16#701,
            LEN      := 0,
            DATAADDR := 0,
            RESPOND  := TRUE
        );
    END_IF
    bClearRead := TRUE;
END_IF

END_PROGRAM

// ---- POUs/P200_CapPreScrewer.TcPOU
PROGRAM P200_CapPreScrewer
VAR_INPUT
	bEnable											: BOOL;	 										// Aktywacja bloku stacji					
	bRun											: BOOL; 
  	bPreRun											: BOOL; 
	bPlacePermission								: BOOL;                  				
	bHoming											: BOOL;                    				
	bManualMode										: BOOL;                     					// Tryb manualny
	bReset											: BOOL; 
	bIgnoreError									: BOOL;                    				
	iStationIndex									: UDINT		:= 1130;							// Numer stacji 
	wsStationName									: WSTRING	:= "Wkładacz zamknięć";		// Nazwa stacji
	stParameters									: ST_CapPreScrewerParameters := (	tTimeVacuumWatchdog		:= T#500MS,
																					lrTopZPosition				:= 400,
																					lrPickZPosition				:= 364,
																					lrPickYPosition				:= 26,
																					lrPlaceZPosition 			:= 236,		
																					lrCartesianCatchZPosition	:= 240,
																					lrPlaceYPosition 			:= 265,
																					lrCapCatcherZPosition 		:= 245,								
																					lrStrawCatcherZPosition 	:= 240,
																					LrCheckStrawCatcherActuatorZPosition:= 238,
																					lrScrewerStartZPosition 	:= 230,
																					lrCapCapCatcherRelese 		:= 228,
																					lrCatcherTopPosition 		:= 150,
																					lrCatcherCatchingPosition 	:= 130,
																					lrCatcherPlacePosition 		:= 70,
																					lrBendingDistance			:= 30,
																					lrScrewDistance				:= 180,
																					lrStrawInsertDistance 		:= 50,
																					lrCatcherSpeed 				:= 15,
																					lrPickerSpeed 				:= 15,
																					lrScrewSpeed 				:= 90,
																					lrCatcherMaxHight			:= 249,
																					lrCatcherMinHight			:= 0,
																					rCatcherHightOffset			:= 250,
																					lrCatcherHightSV			:= 90,	
																					rPulseRatio					:= 0.0140209058,
																					lrCatcherJerk				:= 100_000.0,
																					lrPickerJerk				:= 100_000.0,
																					lrScrewJerk					:= 1_000_000.0,
																					bRejectON					:= TRUE);
	
	
	//Wejścia sprzętowe
	bCapSuckerVacumOk1						: BOOL;		//Sygnał podciśnienia na ssawce nakrętki 1
	bCapSuckerVacumOk2						: BOOL;		//Sygnał podciśnienia na ssawce nakrętki 2
	bCapSuckerVacumOk3						: BOOL;		//Sygnał podciśnienia na ssawce nakrętki 3
	bCapSuckerVacumOk4						: BOOL;		//Sygnał podciśnienia na ssawce nakrętki 4
	
	diCapSuckerVacumOk1				AT%I*	: DINT;
    diCapSuckerVacumOk2				AT%I*	: DINT;
    diCapSuckerVacumOk3				AT%I*	: DINT;
    diCapSuckerVacumOk4				AT%I*	: DINT;

	iCapSuckerVacumOk1				AT%I*	: INT;
    iCapSuckerVacumOk2				AT%I*	: INT;
    iCapSuckerVacumOk3				AT%I*	: INT;
    iCapSuckerVacumOk4				AT%I*	: INT;
	
	
	bStrawCatcherOut		AT	%I*			: BOOL;		//Sygnał z krańcówki - wysunięty łapacz słomek
	bStrawCatcherIn			AT	%I*			: BOOL;		//Sygnał z krańcówki - wysunięty łapacz słomek
	
	bStrawCatcherOpen1		AT	%I*			: BOOL;		//Sygnał z krańcówki - otwart łapacz słomek 1
	bStrawCatcherOpen2		AT	%I*			: BOOL;		//Sygnał z krańcówki - otwart łapacz słomek 2
	bStrawCatcherOpen3		AT	%I*			: BOOL;		//Sygnał z krańcówki - otwart łapacz słomek 3
	bStrawCatcherOpen4		AT	%I*			: BOOL;		//Sygnał z krańcówki - otwart łapacz słomek 4
	
	bPendantDownwardMovement	AT%I*		: BOOL;			// Kaseta sterownicza ruch do góry
	bPendantUpwardMovement		AT%I*		: BOOL; 		// Kaseta sterownicza ruch do dolu
	bPendantUpDownFast			AT%I*		: BOOL;			// Kaseta sterownicza góra/dól- wyższa prędkośc
	bPendantRightwardMovement	AT%I*		: BOOL; 		// Kaseta sterownicza ruch w prawo
	bPendantLeftwardMovement	AT%I*		: BOOL; 		// Kaseta sterownicza ruch w lewo
	bPendantRightLeftFast		AT%I*		: BOOL;			// Kaseta sterownicza lewo/prawo- wyższa prędkośc
	
	bManualBottleGripperUp					: BOOL;
	bManualBottleGripperDown				: BOOL;
	
	bManualCartesianYJogPlus		: BOOL;			//Ruch ręczny podajnika zamknięć 
	bManualCartesianYJogMinus		: BOOL;			//Ruch ręczny podajnika zamknięć 
	bManualCartesianZJogPlus		: BOOL;			//Ruch ręczny podajnika zamknięć 
	bManualCartesianZJogMinus		: BOOL;			//Ruch ręczny podajnika zamknięć 
	
	bManualPreScrewerJogPlus		: BOOL;
	bManualPreScrewerJogMinus		: BOOL;
	
	bManualCatcherJogPlus			: BOOL;
	bManualCatcherJogMinus			: BOOL;
	bSimulationEna					: BOOL;
END_VAR

VAR_OUTPUT
	bBottleGrippers				AT	%Q*		: BOOL;						//Sygnał do zaworu - łapania szyjek butelek

	bCapSucker1					AT	%Q*		: BOOL;						//Sygnał do zaworu - zassij nakrętkę 1
	bCapSucker2					AT	%Q*		: BOOL;						//Sygnał do zaworu - zassij nakrętkę 2
	bCapSucker3					AT	%Q*		: BOOL;						//Sygnał do zaworu - zassij nakrętkę 3
	bCapSucker4					AT	%Q*		: BOOL;						//Sygnał do zaworu - zassij nakrętkę 4
	
	bCapBlower1					AT	%Q*		: BOOL;						//Sygnał do zaworu - wydmuchaj nakrętkę 1
	bCapBlower2					AT	%Q*		: BOOL;						//Sygnał do zaworu - wydmuchaj nakrętkę 2
	bCapBlower3					AT	%Q*		: BOOL;						//Sygnał do zaworu - wydmuchaj nakrętkę 3
	bCapBlower4					AT	%Q*		: BOOL;						//Sygnał do zaworu - wydmuchaj nakrętkę 4
	
	bCapCatcher1				AT	%Q*		: BOOL;						//Sygnał do zaworu - złap nakrętkę 1
	bCapCatcher2				AT	%Q*		: BOOL;						//Sygnał do zaworu - złap nakrętkę 2
	bCapCatcher3				AT	%Q*		: BOOL;						//Sygnał do zaworu - złap nakrętkę 3
	bCapCatcher4				AT	%Q*		: BOOL;						//Sygnał do zaworu - złap nakrętkę 4
	
	bStrawCatchersOpen			AT	%Q*		: BOOL;						//Sygnał do zaworu - otwórz chwytaki słomek
	bStrawCatchersClose			AT	%Q*		: BOOL;						//Sygnał do zaworu - zamknij chwytaki słomek
	
	bStrawCatcherActuatorOut	AT	%Q*		: BOOL;						//Sygnał do zaworu - wysuń łapacz słomek
	bStrawCatcherActuatorIn		AT	%Q*		: BOOL;						//Sygnał do zaworu - wsuń łapacz słomek
	
	
	eState									: E_Station;								// Stan ogólny bloku
	eRunnigState							: E_CapPreScrewer;
	bError									: BOOL;										// Błąd bloku
	udiErrorID								: UDINT;									// Numer błędu
	sErrorDescription1						: STRING(200);								// Opis błędu 1
	sErrorDescription2						: STRING(200);								// Opis błędu 2
	sErrorStationName						: STRING;									// Nazwa stacji
	bHomingDone								: BOOL;										// Stacja zbazowana
	bCycleNotDone							: BOOL;										// Cykl nie został wykonany
	bCycleDone								: BOOL;										// Cykl został wykonany
	aCapPresence							: ARRAY [1..4] OF BOOL;
	bAnyCapSucker							: BOOL;										//Przynajmniej jedna nakrętka pobrana
	bRejectDone								: BOOL;
END_VAR



VAR
	fbCapPreScrewer							: FB_CapPreScrewer;
	fbCapPreScrewerState					: FB_State;
	
	bTestRun								: BOOL;
	bTestHoming								: BOOL;
	bTestReset								: BOOL;
	
	tonCheckVacuum							: TON;
	tCycleTime								: TIME;
	bMissingCaps							: BOOL;

	bCartesianSafePos						: BOOL;
	stCommandsIN							: ST_CapPreScrewerCommandsIn;
	bTestEnable: BOOL;
	bCapSuckerTemp: ARRAY [1..4] OF  BOOL;
	bVacuumTest: BOOL;
	bTestPreRun: BOOL;
	tonCapCatcher1	: TON;
	tonCapCatcher2	: TON;
	tonCapCatcher3	: TON;
	tonCapCatcher4	: TON;
	fbVacuumInputFilter	: ARRAY [1..4] OF FB_FilterEx;
	bTestSettingStation	: BOOL;
	ftTestSettingStation	: F_TRIG;
	fbTimeFilter	: FB_DigitalInput_1;
END_VAR



IF bCapSucker4 AND NOT bCapSuckerVacumOk4 AND eState = E_Station.eRunning  THEN
	tCycleTime			:= tonCheckVacuum.ET;
END_IF

tonCheckVacuum(IN := bCapSucker4 AND NOT bCapSuckerVacumOk4, PT := T#2D);

GVL_VIS.bCapSorterPreScrewerCatcherStationHeightSet := SEL((ABS(GVL_VIS.lrCapSorterPreScrewerCatcherStationHeightCV-GVL_Recipe.lrCapSorterPreScrewerCatcherHightSVShow)<=1.0),
													GVL_VIS.bCapSorterPreScrewerCatcherStationHeightSet, FALSE);

//*****************Sterowanie zaworami ssawek***********************************
bCapSucker1 := NOT stparameters.bvacuumDeactivate AND bCapSuckerTemp[1];
bCapSucker2 := NOT stparameters.bvacuumDeactivate AND bCapSuckerTemp[2];
bCapSucker3 := NOT stparameters.bvacuumDeactivate AND bCapSuckerTemp[3];
bCapSucker4 := NOT stparameters.bvacuumDeactivate AND bCapSuckerTemp[4];

stParameters.LrCheckStrawCatcherActuatorZPosition;
stParameters.lrStrawCatcherZPosition;
stParameters.lrCartesianCatchZPosition;

//bAnyCapSucker := bCapSucker1 OR bCapSucker2 OR bCapSucker3 OR bCapSucker4;
//fbCapPreScrewer.stMoverStatus := SEL(P190_CapFeeder.stMover1Status.bInPlacePosition, P190_CapFeeder.stMover2Status, P190_CapFeeder.stMover1Status);

//_____________________Generowanie stanu do wizki______________________________________
fbCapPreScrewerState(	eState 					:= eState,
			 			bRun					:= bRun,
			 			sStateDesc				=> GVL_VIS.sCapSorterPreScrewerState,
			 			iState					=> GVL_VIS.iCapSorterPreScrewerState);
				
stParameters.lrPickerSpeedWhenScrewer;

ACT_FB();

//Adresy dla komunikacji ADS
stParameters.sADS_NetId					:= '192.168.40.160.4.1';
stParameters.nAxisY_ADS_SlaveAddr		:= 1020;
stParameters.nAxisZ_ADS_SlaveAddr		:= 1020;
stParameters.nCatcher_ADS_SlaveAddr		:= 1019;


//Przepisanie zmiennych
stCommandsIN.bPendantDownwardMovement	:= bPendantDownwardMovement	;
stCommandsIN.bPendantUpwardMovement		:= bPendantUpwardMovement	;	
stCommandsIN.bPendantUpDownFast			:= bPendantUpDownFast		;	
stCommandsIN.bPendantRightwardMovement	:= bPendantRightwardMovement;	
stCommandsIN.bPendantLeftwardMovement	:= bPendantLeftwardMovement	;
stCommandsIN.bPendantRightLeftFast		:= bPendantRightLeftFast	;	
//stCommandsIN.bChoseRecipe				:= GVL_Communication.bChooseRecipe;


GVL_Recipe.lrCapSorterPreScrewerPickXMover1PositionShow			;
GVL_recipe.lrCapSorterPreScrewerPlaceXPositionShow			;
GVL_recipe.lrCapSorterPreScrewerTopZPositionShow			;
GVL_recipe.lrCapSorterPreScrewerPickZPositionShow			;
GVL_recipe.lrCapSorterPreScrewerCatcherCatchingPositionShow	;
GVL_recipe.lrCapSorterPreScrewerCartesianCatchZPositionShow;
GVL_recipe.LrCapSorterPreScrewerCheckStrawCatcherActuatorZPosition;
GVL_recipe.lrCapSorterPreScrewerPlaceZPositionShow			;
GVL_recipe.lrCapSorterPreScrewerCapCatcherZPositionShow		;
GVL_recipe.lrCapSorterPreScrewerGripperOpenPositionShow		;
GVL_recipe.lrCapSorterPreScrewerCatcherReleseShow			;
GVL_recipe.lrCapSorterPreScrewerStrawCatcherZPositionShow	;
GVL_recipe.lrCapSorterPreScrewerScrewerStartZPositionShow	;
GVL_recipe.lrCapSorterPreScrewerBendingDistanceShow			;
                                                            
GVL_Recipe.lrCapSorterPreScrewerCatcherHightSVShow			;
GVL_Recipe.lrCapSorterPreScrewerCatcherCatchingPositionShow	;
GVL_Recipe.lrCapSorterPreScrewerCatcherPlacePositionShow	;
                                                            
GVL_recipe.lrCapSorterPreScrewerScrewDistanceShow			;
GVL_recipe.lrCapSorterPreScrewerStrawInsertDistance			;
                                                            
GVL_Recipe.lrCapSorterPreScrewerCatcherSpeedShow			;
GVL_Recipe.lrCapSorterPreScrewerPickerSpeedShow				;
GVL_Recipe.lrCapSorterPreScrewerScrewSpeedShow				;
                                                            
GVL_Recipe.lrCapSorterPreScrewerCatcherHightSVShow			;


stParameters.bPickerActiv[1];

stParameters.rCatcherHightOffset ;

// bCapSuckerVacumOk1			:= ABS(diCapSuckerVacumOk1) >= 450;	
// bCapSuckerVacumOk2			:= ABS(diCapSuckerVacumOk2) >= 450;	
// bCapSuckerVacumOk3			:= ABS(diCapSuckerVacumOk3) >= 450;	
// bCapSuckerVacumOk4			:= ABS(diCapSuckerVacumOk4) >= 450;	
fbVacuumInputFilter[1](rIn := INT_TO_REAL(iCapSuckerVacumOk1), tTimeConstant	:= T#25MS);
fbVacuumInputFilter[2](rIn := INT_TO_REAL(iCapSuckerVacumOk2), tTimeConstant	:= T#25MS);
fbVacuumInputFilter[3](rIn := INT_TO_REAL(iCapSuckerVacumOk3), tTimeConstant	:= T#25MS);
fbVacuumInputFilter[4](rIn := INT_TO_REAL(iCapSuckerVacumOk4), tTimeConstant	:= T#25MS);


GVL_VIS.lrCapSorterPreScrewerVacuumLevel_1	:= DINT_TO_LREAL(iCapSuckerVacumOk1)/10_000;
GVL_VIS.lrCapSorterPreScrewerVacuumLevel_2	:= DINT_TO_LREAL(iCapSuckerVacumOk2)/10_000;
GVL_VIS.lrCapSorterPreScrewerVacuumLevel_3	:= DINT_TO_LREAL(iCapSuckerVacumOk3)/10_000;
GVL_VIS.lrCapSorterPreScrewerVacuumLevel_4	:= DINT_TO_LREAL(iCapSuckerVacumOk4)/10_000;

bCapSuckerVacumOk1			:= ABS(iCapSuckerVacumOk1/10) >= 480;	
bCapSuckerVacumOk2			:= ABS(iCapSuckerVacumOk2/10) >= 480;	
bCapSuckerVacumOk3			:= ABS(iCapSuckerVacumOk3/10) >= 480;	
bCapSuckerVacumOk4			:= ABS(iCapSuckerVacumOk4/10) >= 480;	

tonCapCatcher1(IN := bCapCatcher1, PT := T#100MS);
tonCapCatcher2(IN := bCapCatcher2, PT := T#100MS);
tonCapCatcher3(IN := bCapCatcher3, PT := T#100MS);
tonCapCatcher4(IN := bCapCatcher4, PT := T#100MS);




IF bTestSettingStation THEN
	IF GVL_VIS.lrCapSorterPreScrewerCatcherStationHeightCV < 300 AND NOT GVL_VIS.bCapSorterPreScrewerCatcherStationDown THEN
		fbTimeFilter.In	:= TRUE;
		GVL_VIS.bCapSorterPreScrewerCatcherStationUp	:= fbTimeFilter.bIn;
	ELSIF GVL_VIS.lrCapSorterPreScrewerCatcherStationHeightCV >= 300 THEN
		fbTimeFilter.In	:= FALSE;
		GVL_VIS.bCapSorterPreScrewerCatcherStationUp	:= FALSE;
		GVL_VIS.bCapSorterPreScrewerCatcherStationDown 	S= NOT fbTimeFilter.bIn;
	ELSIF GVL_VIS.lrCapSorterPreScrewerCatcherStationHeightCV <= 100 THEN
		GVL_VIS.bCapSorterPreScrewerCatcherStationDown 	:= FALSE;	
	END_IF	
ELSIF ftTestSettingStation.Q THEN
	fbTimeFilter.In	:= FALSE;
	GVL_VIS.bCapSorterPreScrewerCatcherStationUp	:= FALSE;
	GVL_VIS.bCapSorterPreScrewerCatcherStationDown 	:= FALSE;		
END_IF

fbTimeFilter.tTimeOn 	:= T#500MS;
fbTimeFilter.tTimeOff	:= T#500mS;
fbTimeFilter.FilterTrig();
ftTestSettingStation(CLK := bTestSettingStation);

ACTION ACT_FB:
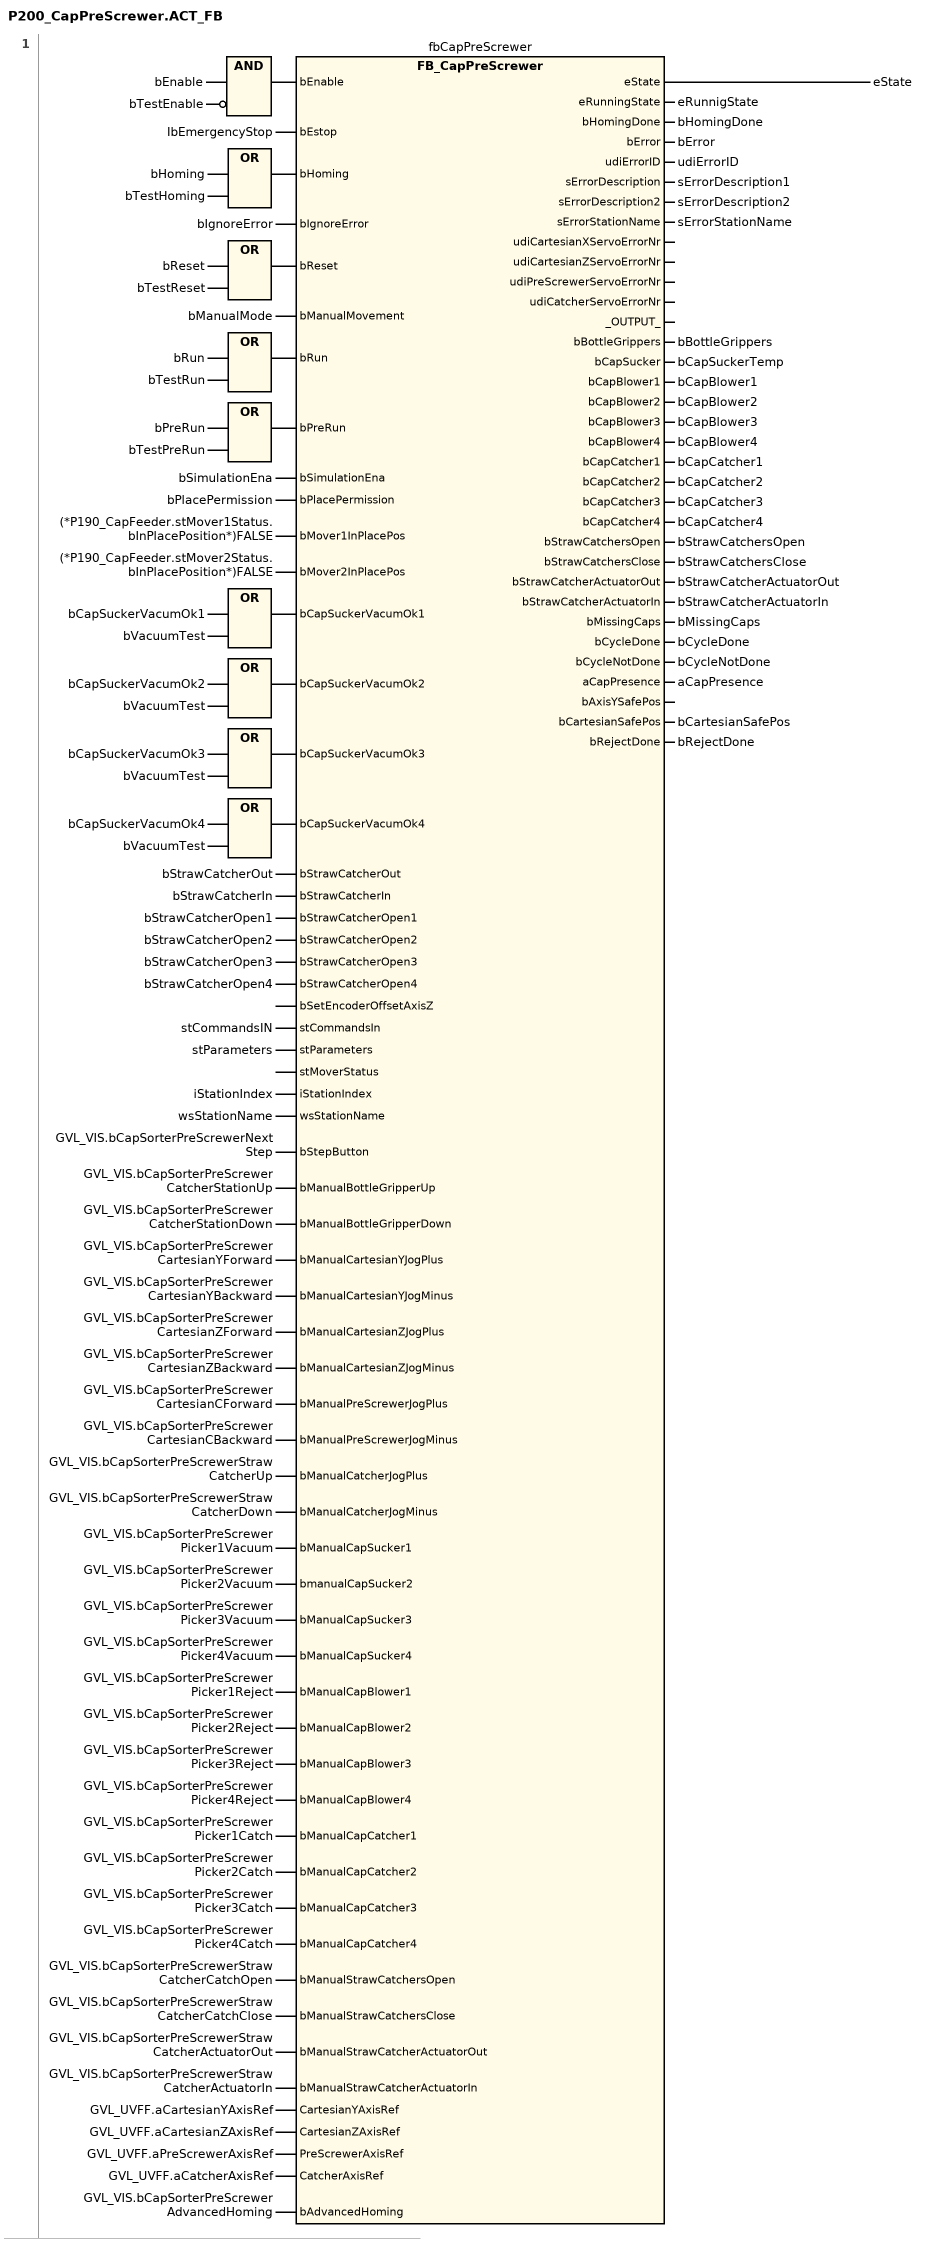
// NETWORK 1
fbCapPreScrewer(
    bEnable := bEnable AND NOT bTestEnable,
    bEstop := IbEmergencyStop,
    bHoming := bHoming OR bTestHoming,
    bIgnoreError := bIgnoreError,
    bReset := bReset OR bTestReset,
    bManualMovement := bManualMode,
    bRun := bRun OR bTestRun,
    bPreRun := bPreRun OR bTestPreRun,
    bSimulationEna := bSimulationEna,
    bPlacePermission := bPlacePermission,
    bMover1InPlacePos := (*P190_CapFeeder.stMover1Status.bInPlacePosition*)FALSE,
    bMover2InPlacePos := (*P190_CapFeeder.stMover2Status.bInPlacePosition*)FALSE,
    bCapSuckerVacumOk1 := bCapSuckerVacumOk1 OR bVacuumTest,
    bCapSuckerVacumOk2 := bCapSuckerVacumOk2 OR bVacuumTest,
    bCapSuckerVacumOk3 := bCapSuckerVacumOk3 OR bVacuumTest,
    bCapSuckerVacumOk4 := bCapSuckerVacumOk4 OR bVacuumTest,
    bStrawCatcherOut := bStrawCatcherOut,
    bStrawCatcherIn := bStrawCatcherIn,
    bStrawCatcherOpen1 := bStrawCatcherOpen1,
    bStrawCatcherOpen2 := bStrawCatcherOpen2,
    bStrawCatcherOpen3 := bStrawCatcherOpen3,
    bStrawCatcherOpen4 := bStrawCatcherOpen4,
    stCommandsIn := stCommandsIN,
    stParameters := stParameters,
    iStationIndex := iStationIndex,
    wsStationName := wsStationName,
    bStepButton := GVL_VIS.bCapSorterPreScrewerNextStep,
    bManualBottleGripperUp := GVL_VIS.bCapSorterPreScrewerCatcherStationUp,
    bManualBottleGripperDown := GVL_VIS.bCapSorterPreScrewerCatcherStationDown,
    bManualCartesianYJogPlus := GVL_VIS.bCapSorterPreScrewerCartesianYForward,
    bManualCartesianYJogMinus := GVL_VIS.bCapSorterPreScrewerCartesianYBackward,
    bManualCartesianZJogPlus := GVL_VIS.bCapSorterPreScrewerCartesianZForward,
    bManualCartesianZJogMinus := GVL_VIS.bCapSorterPreScrewerCartesianZBackward,
    bManualPreScrewerJogPlus := GVL_VIS.bCapSorterPreScrewerCartesianCForward,
    bManualPreScrewerJogMinus := GVL_VIS.bCapSorterPreScrewerCartesianCBackward,
    bManualCatcherJogPlus := GVL_VIS.bCapSorterPreScrewerStrawCatcherUp,
    bManualCatcherJogMinus := GVL_VIS.bCapSorterPreScrewerStrawCatcherDown,
    bManualCapSucker1 := GVL_VIS.bCapSorterPreScrewerPicker1Vacuum,
    bmanualCapSucker2 := GVL_VIS.bCapSorterPreScrewerPicker2Vacuum,
    bManualCapSucker3 := GVL_VIS.bCapSorterPreScrewerPicker3Vacuum,
    bManualCapSucker4 := GVL_VIS.bCapSorterPreScrewerPicker4Vacuum,
    bManualCapBlower1 := GVL_VIS.bCapSorterPreScrewerPicker1Reject,
    bManualCapBlower2 := GVL_VIS.bCapSorterPreScrewerPicker2Reject,
    bManualCapBlower3 := GVL_VIS.bCapSorterPreScrewerPicker3Reject,
    bManualCapBlower4 := GVL_VIS.bCapSorterPreScrewerPicker4Reject,
    bManualCapCatcher1 := GVL_VIS.bCapSorterPreScrewerPicker1Catch,
    bManualCapCatcher2 := GVL_VIS.bCapSorterPreScrewerPicker2Catch,
    bManualCapCatcher3 := GVL_VIS.bCapSorterPreScrewerPicker3Catch,
    bManualCapCatcher4 := GVL_VIS.bCapSorterPreScrewerPicker4Catch,
    bManualStrawCatchersOpen := GVL_VIS.bCapSorterPreScrewerStrawCatcherCatchOpen,
    bManualStrawCatchersClose := GVL_VIS.bCapSorterPreScrewerStrawCatcherCatchClose,
    bManualStrawCatcherActuatorOut := GVL_VIS.bCapSorterPreScrewerStrawCatcherActuatorOut,
    bManualStrawCatcherActuatorIn := GVL_VIS.bCapSorterPreScrewerStrawCatcherActuatorIn,
    CartesianYAxisRef := GVL_UVFF.aCartesianYAxisRef,
    CartesianZAxisRef := GVL_UVFF.aCartesianZAxisRef,
    PreScrewerAxisRef := GVL_UVFF.aPreScrewerAxisRef,
    CatcherAxisRef := GVL_UVFF.aCatcherAxisRef,
    bAdvancedHoming := GVL_VIS.bCapSorterPreScrewerAdvancedHoming,
    eRunningState => eRunnigState,
    bHomingDone => bHomingDone,
    bError => bError,
    udiErrorID => udiErrorID,
    sErrorDescription => sErrorDescription1,
    sErrorDescription2 => sErrorDescription2,
    sErrorStationName => sErrorStationName,
    bBottleGrippers => bBottleGrippers,
    bCapSucker => bCapSuckerTemp,
    bCapBlower1 => bCapBlower1,
    bCapBlower2 => bCapBlower2,
    bCapBlower3 => bCapBlower3,
    bCapBlower4 => bCapBlower4,
    bCapCatcher1 => bCapCatcher1,
    bCapCatcher2 => bCapCatcher2,
    bCapCatcher3 => bCapCatcher3,
    bCapCatcher4 => bCapCatcher4,
    bStrawCatchersOpen => bStrawCatchersOpen,
    bStrawCatchersClose => bStrawCatchersClose,
    bStrawCatcherActuatorOut => bStrawCatcherActuatorOut,
    bStrawCatcherActuatorIn => bStrawCatcherActuatorIn,
    bMissingCaps => bMissingCaps,
    bCycleDone => bCycleDone,
    bCycleNotDone => bCycleNotDone,
    aCapPresence => aCapPresence,
    bCartesianSafePos => bCartesianSafePos,
    bRejectDone => bRejectDone); // FB_CapPreScrewer
eState := fbCapPreScrewer.eState;
END_ACTION

END_PROGRAM

// ---- POUs/FB/FB_CapPreScrewer.TcPOU
FUNCTION_BLOCK FB_CapPreScrewer
VAR_INPUT
	bEnable								: BOOL;		//Zezwolenie na pracę
	bEstop								: BOOL;		//Stop awaryjny nieaktywny
	bHoming								: BOOL;		//Zezwolenie na wykonanie bazowania
	bIgnoreError						: BOOL;		//Ignorowania błędów cyklu pracy
	
	bReset								: BOOL;		//Reset błędu, jeśli w stanie "eError
	bManualMovement						: BOOL;		//Zezwolenie na ruchy ręcznę
	
	bRun								: BOOL;		//Rozkaz uruchomienia zakręcarki
	bPreRun								: BOOL;		//Przygotowanie stacji do pracy
	bSimulationEna						: BOOL;		//Tryb symulacji
	bPlacePermission					: BOOL;		//Zezwolenenie na wkładanie nakrentki w butelkę
	bMover1InPlacePos					: BOOL;		//Wózek 1 na pozycji Place
	bMover2InPlacePos					: BOOL;		//Wózek 2 na pozycji Place

	bCapSuckerVacumOk1					: BOOL;		//Sygnał podciśnienia na ssawce nakrętki 1
	bCapSuckerVacumOk2					: BOOL;		//Sygnał podciśnienia na ssawce nakrętki 2
	bCapSuckerVacumOk3					: BOOL;		//Sygnał podciśnienia na ssawce nakrętki 3
	bCapSuckerVacumOk4					: BOOL;		//Sygnał podciśnienia na ssawce nakrętki 4
	
	bStrawCatcherOut					: BOOL;		//Sygnał z krańcówki - wysunięty łapacz słomek
	bStrawCatcherIn						: BOOL;		//Sygnał z krańcówki - wysunięty łapacz słomek
	
	bStrawCatcherOpen1					: BOOL;		//Sygnał z krańcówki - otwart łapacz słomek 1
	bStrawCatcherOpen2					: BOOL;		//Sygnał z krańcówki - otwart łapacz słomek 2
	bStrawCatcherOpen3					: BOOL;		//Sygnał z krańcówki - otwart łapacz słomek 3
	bStrawCatcherOpen4					: BOOL;		//Sygnał z krańcówki - otwart łapacz słomek 4
	bSetEncoderOffsetAxisZ				: BOOL;		//Ustaw pozycję enkodera osi Z 
	
	stCommandsIn						: ST_CapPreScrewerCommandsIn;		

	stParameters						: ST_CapPreScrewerParameters;
	stMoverStatus						: ST_MoverState;
	
	iStationIndex						: UDINT;		//Numer stacji 
	wsStationName						: WSTRING;	//Nazwa stacji
	
END_VAR

VAR_OUTPUT
	eState							: E_Station;			//Stan ogólny bloku
	eRunningState					: E_CapPreScrewer; 		//Stan załapywarki
	bHomingDone						: BOOL;					//Stacja zbazowana
	bError							: BOOL;						//Błąd stacji
	udiErrorID						: UDINT;					//Nr błędu zakręcarki
	sErrorDescription				: STRING(200);				//Opis błędu
	sErrorDescription2				: STRING(200);				//Opis błędu
	sErrorStationName				: STRING;					//Nazwa stacj
	
	udiCartesianXServoErrorNr		: UDINT;					//Nr błędu serwa poziomego X
	udiCartesianZServoErrorNr		: UDINT;					//Nr błędu serwa pionowego Y
	udiPreScrewerServoErrorNr		: UDINT;					//Nr błędu serwa obrotowego załapywarki
	udiCatcherServoErrorNr			: UDINT;					//Nr błędu serwo pionowego uchwytu słomek
	
	_OUTPUT_						: BOOL;
	bBottleGrippers					: BOOL;						//Sygnał do zaworu - łapania szyjek butelek

	bCapSucker 						: ARRAY [1..4] OF BOOL;		//Sygnał do zaworu - zassij nakrętkę
	//bCapSucker2						: BOOL;						//Sygnał do zaworu - zassij nakrętkę 2
	//bCapSucker3						: BOOL;						//Sygnał do zaworu - zassij nakrętkę 3
	//bCapSucker4						: BOOL;						//Sygnał do zaworu - zassij nakrętkę 4
	
	bCapBlower1						: BOOL;						//Sygnał do zaworu - wydmuchaj nakrętkę 1
	bCapBlower2						: BOOL;						//Sygnał do zaworu - wydmuchaj nakrętkę 2
	bCapBlower3						: BOOL;						//Sygnał do zaworu - wydmuchaj nakrętkę 3
	bCapBlower4						: BOOL;						//Sygnał do zaworu - wydmuchaj nakrętkę 4
	
	bCapCatcher1					: BOOL;						//Sygnał do zaworu - złap nakrętkę 1
	bCapCatcher2					: BOOL;						//Sygnał do zaworu - złap nakrętkę 2
	bCapCatcher3					: BOOL;						//Sygnał do zaworu - złap nakrętkę 3
	bCapCatcher4					: BOOL;						//Sygnał do zaworu - złap nakrętkę 4
	
	bStrawCatchersOpen				: BOOL;						//Sygnał do zaworu - otwórz chwytaki słomek
	bStrawCatchersClose				: BOOL;						//Sygnał do zaworu - zamknij chwytaki słomek
	
	bStrawCatcherActuatorOut		: BOOL;						//Sygnał do zaworu - wysuń łapacz słomek
	bStrawCatcherActuatorIn			: BOOL;						//Sygnał do zaworu - wsuń łapacz słomek
	bMissingCaps					: BOOL;						//Żadna nakretka nie zostala pobrana
	
	bCycleDone						: BOOL;						//Cykl zakończono
	bCycleNotDone					: BOOL;						//Nie zakończono cyklu przestawiania wózków
	aCapPresence					: ARRAY [1..4] OF BOOL;		//jakie nakretki zostaly odlozone do butelek
	bAxisYSafePos					: BOOL;						//Bezpieczna pozycja osi Y dla przejazdu mówerów
	bCartesianSafePos				: BOOL;						//Bezpieczna pozycja kartezjana dla przejazdu mówerów
	bRejectDone						: BOOL;						// Zakończony odrzut
END_VAR

VAR_IN_OUT
	bStepButton						: BOOL; 		//Następny krok sekwencji	

	bManualBottleGripperUp			: BOOL;			//Ręczny ruch Jisang
	bManualBottleGripperDown		: BOOL;			//Ręczny ruch Jisang
	
	bManualCartesianYJogPlus		: BOOL;			//Ruch ręczny podajnika zamknięć 
	bManualCartesianYJogMinus		: BOOL;			//Ruch ręczny podajnika zamknięć 
	bManualCartesianZJogPlus		: BOOL;			//Ruch ręczny podajnika zamknięć 
	bManualCartesianZJogMinus		: BOOL;			//Ruch ręczny podajnika zamknięć 
	
	bManualPreScrewerJogPlus		: BOOL;
	bManualPreScrewerJogMinus		: BOOL;
	
	bManualCatcherJogPlus			: BOOL;
	bManualCatcherJogMinus			: BOOL;

	bManualCapSucker1				: BOOL;						//Ręczne sterowanie zaworu - zassij nakrętkę 1
	bmanualCapSucker2				: BOOL;						//Ręczne sterowanie - zassij nakrętkę 2
	bManualCapSucker3				: BOOL;						//Ręczne sterowanie - zassij nakrętkę 3
	bManualCapSucker4				: BOOL;						//Ręczne sterowanie - zassij nakrętkę 4
	                                
	bManualCapBlower1				: BOOL;						//Ręczne sterowanie - wydmuchaj nakrętkę 1
	bManualCapBlower2				: BOOL;						//Ręczne sterowanie - wydmuchaj nakrętkę 2
	bManualCapBlower3				: BOOL;						//Ręczne sterowanie - wydmuchaj nakrętkę 3
	bManualCapBlower4				: BOOL;						//Ręczne sterowanie - wydmuchaj nakrętkę 4
	
	bManualCapCatcher1				: BOOL;						//Ręczne sterowanie - złap nakrętkę 1
	bManualCapCatcher2				: BOOL;						//Ręczne sterowanie - złap nakrętkę 2
	bManualCapCatcher3				: BOOL;						//Ręczne sterowanie - złap nakrętkę 3
	bManualCapCatcher4				: BOOL;						//Ręczne sterowanie - złap nakrętkę 4
	
	bManualStrawCatchersOpen		: BOOL;						//Ręczne sterowanie - zamknij chwytaki słomek
	bManualStrawCatchersClose		: BOOL;                     //Ręczne sterowanie - otwórz chwytaki słomek
	                                  
	bManualStrawCatcherActuatorOut	: BOOL;						//Ręczne sterowanie - wysuń łapacz słomek
	bManualStrawCatcherActuatorIn	: BOOL;                     //Ręczne sterowanie - wsuń łapacz słomek
	
	CartesianYAxisRef				: AXIS_REF;		//Struktura sterowania NC dla serwa przesuwania poziomego
	CartesianZAxisRef				: AXIS_REF;		//Struktura sterowania NC dla serwa przesuwania pionowego
	PreScrewerAxisRef				: AXIS_REF;		//Struktura sterowania NC dla serwa załapywania nakrętek
	CatcherAxisRef					: AXIS_REF;		//Struktura sterowania NC dla serwa prowadzenia słomki
	bAdvancedHoming: BOOL;
END_VAR

VAR
	fbStrawCatcherLift				: FB_Checker;

	diMover1VacuumRetry				: ARRAY [1..4] OF DINT;					// Ilość prób pobrania wózek 1, słoty 1..4
	diMover2VacuumRetry				: ARRAY [1..4] OF DINT;					// Ilość prób pobrania wózek 2, słoty 1..4
	
	tonDelayServoOn					: TON;
	
	mcCartesianYManualMove			: MC_JOG; 			// Blok ruchu ręcznego 
	mcCartesianZManualMove			: MC_JOG; 			// Blok ruchu ręcznego
	mcPreScrewerManualMove			: MC_JOG; 			// Blok ruchu ręcznego
	mcCatcherManualMove				: MC_JOG; 			// Blok ruchu ręcznego
	
	mcCartesianYStop				: MC_Stop;			// Trwałe zatrzymywanie Serwo
	mcCartesianZStop				: MC_Stop;			// Trwałe zatrzymywanie Serwo
	mcPreScrewerStop				: MC_Stop;			// Trwałe zatrzymywanie Serwo
	mcCatcherStop					: MC_Stop;			// Trwałe zatrzymywanie Serwo
	
	mcCatcherHalt				: MC_Halt;			// Trwałe zatrzymywanie Serwo
	
//	mcMover1MoveVelocity		: MC_MoveVelocity;		// Ruch prędkościowy
//	mcMover2MoveVelocity		: MC_MoveVelocity;		// Ruch prędkościowy
//	mcMover1MoveVelocity2		: MC_MoveVelocity;		// Ruch prędkościowy
//	mcMover2MoveVelocity2		: MC_MoveVelocity;		// Ruch prędkościowy	
//	mcMover1MoveRelative		: MC_MoveRelative; 		// Ruch relatywny
	
	mcCartesianYMoveAbsolute	: MC_MoveAbsolute; 		// Ruch absolutny
	mcCartesianYMoveRelative	: MC_MoveRelative;		// Ruch względny
	mcCartesianZMoveAbsolute	: MC_MoveAbsolute; 		// Ruch absolutny
	mcCartesianZMoveAbsolute2	: MC_MoveAbsolute; 		// Ruch absolutny
	mcPreScrewerMoveAbsolute	: MC_MoveAbsolute; 		// Ruch absolutny
	mcPreScrewerMoveRelative	: MC_MoveRelative; 		// Ruch względny
	mcCatcherMoveAbsolute		: MC_MoveAbsolute; 		// Ruch absolutny
	
	fbAxisYPositioningOffset	: FB_CoEAX8000SetPositionOffset;
	fbAxisZPositioningOffset	: FB_CoEAX8000SetPositionOffset;
	
	mcCartesianYPower			: MC_Power;			 	// Zasilanie napędu
	mcCartesianZPower			: MC_Power;			 	// Zasilanie napędu
	mcPreScrewerPower			: MC_Power;			 	// Zasilanie napędu
	mcCatcherPower				: MC_Power;			 	// Zasilanie napędu
	
	mcPreScrewerHome			: MC_Home;	
	
	bCartesianYServoPower		: BOOL;					// Zmienna sterujaca zasilaniem serwo
	bCartesianZServoPower		: BOOL;					// Zmienna sterujaca zasilaniem serwo	
	bPreScrewerPower			: BOOL;					// Zmienna sterujaca zasilaniem serwo
	bCatcherPower				: BOOL;					// Zmienna sterujaca zasilaniem serwo
	
	fbCartesianYHardReset		: FB_SoEReset; 			// Blok twardego resetu serwa
	fbCartesianZHardReset		: FB_SoEReset; 			// Blok twardego resetu serwa
	fbPreScrewerHardReset		: FB_SoEReset; 			// Blok twardego resetu serwa
	fbCatcherHardReset			: FB_SoEReset; 			// Blok twardego resetu serwa
	mcCartesianYSoftReset		: MC_Reset; 			// blok łagodnego resetu serwa 
	mcCartesianZSoftReset		: MC_Reset; 			// blok łagodnego resetu serwa
	mcPreScrewerSoftReset		: MC_Reset; 			// blok łagodnego resetu serwa
	mcCatcherSoftReset			: MC_Reset; 			// blok łagodnego resetu serwa
	
	(*Bledy, Resetowanie*)
	tonResetting						: TON;
	rtResetCommands						: R_TRIG;
	tonActualMotor1TemperatureTooHigh	: TON;
	tonActualMotor2TemperatureTooHigh	: TON;
		
	bStateError							: BOOL;
	
	eLastState					: E_Station;			// Stan ogólny bloku
	eLastRunningState			: E_CapPreScrewer;		// Stan podbloku
	eLastStateTemp				: E_Station;			// Stan ogólny bloku
	//eLastRunningStateTemp		: E_CapFeeder;		// Stan podbloku
	
	(*Casy od różnych stanów*)
	iAbortingCASE				: INT;
	iStoppingCase 				: INT;
	iHomingCase					: INT;
	iErrorResseting2			: INT;
	iTestResetting				: INT;
	iCountAborting				: INT;
	
	(*Filtry czujników*)
	tonSuckedOk					: ARRAY [1..4] OF TON;
	//tonSuckedOk2				: TON;
	//tonSuckedOk3				: TON;
	//tonSuckedOk4				: TON;
	
	tonStrawCatcherIn			: TON;
	tonStrawCatcherOut			: TON;
	
	tonStrawCatcher1Open		: TON;
	tonStrawCatcher2Open		: TON;
	tonStrawCatcher3Open		: TON;
	tonStrawCatcher4Open		: TON;
	
	tonStrawCatcher1Close		: TON;
	tonStrawCatcher2Close		: TON;
	tonStrawCatcher3Close		: TON;
	tonStrawCatcher4Close		: TON;
	
	//Czasówki do obsługi błędów siłowników
	tonErrorStrawCatcherIn		: TON;
	tonErrorStrawCatcherOut		: TON;
	
	tonErrorStrawCatcherOpen1	: TON;
	tonErrorStrawCatcherOpen2	: TON;
	tonErrorStrawCatcherOpen3	: TON;
	tonErrorStrawCatcherOpen4	: TON;
	
	//Czasówki do obsługi problemu z zasysaniem
	tonErrorSuckerVacum1		: TON;
	tonErrorSuckerVacum2		: TON;
	tonErrorSuckerVacum3		: TON;
	tonErrorSuckerVacum4		: TON;
	tonCapCatcher				: TON;
	
	tonBlowOFF					: TON;
	bCapsBlowON					: BOOL;
	
	tonVacuumWatchdog			: TON;
	i: INT;
	
	tonBlowerON				: ARRAY [1..4] OF TON;	//Cap blowing timers
		
	tonPlacePermission			: TON;
	rtPlacePermission			: R_TRIG;
	bGripperOpen: BOOL;
	bStopAllowed: BOOL;
	
//	fbBottleCatch									: fb
	eBottleCatch1State								:E_Station; 						// Stan chwytaka stabilizujšcego pod podajnikiem nakrętek
	eBottleCatch2State								:E_Station; 						// Stan chwytaka stabilizujšcego pod podajnikiem nakrętek
	eBottleCatch3State								:E_Station; 						// Stan chwytaka stabilizujšcego pod podajnikiem nakrętek
	eBottleCatch4State								:E_Station; 						// Stan chwytaka stabilizujšcego pod podajnikiem nakrętek
	eBottleCatch1RunningState						:E_CatchStationState; 				// Poprzedni stan chwytaka pod podajnikiem nakrętek
	eBottleCatch2RunningState						:E_CatchStationState; 				// Poprzedni stan chwytaka pod podajnikiem nakrętek
	eBottleCatch3RunningState						:E_CatchStationState; 				// Poprzedni stan chwytaka pod podajnikiem nakrętek
	eBottleCatch4RunningState						:E_CatchStationState; 				// Poprzedni stan chwytaka pod podajnikiem nakręte
	fbBottleCatch1State								:FB_State;
	fbBottleCatch2State								:FB_State;
	fbBottleCatch3State								:FB_State;
	fbBottleCatch4State								:FB_State;
	
	IbBottleCatchHeightMotorEncoderPulse			: BOOL;									// Sygnał impulsów enkodera siłownika	
                                            
                                                    
    QbBottleCatchHeightUpCmd              			: BOOL;  								// Zmienna sterownika bezpośrednio sterująca siłownikiem w górę 
    QbBottleCatchHeightDownCmd            			: BOOL;									// Zmienna sterownika bezpośrednio sterująca siłownikiem w dół 	
	bBottleCatcherCatchTemp							: BOOL;
	rtRun											: R_TRIG;
	bTestStrawCatcher								: BOOL;
	bTestError										: BOOL;
	bCatcHActuator1									: BOOL;
	bCatcHActuator2									: BOOL;
	bCatcHActuator3									: BOOL;
	bCatcHActuator4									: BOOL;
                                                	
	bCollisionWithMoverArea							: BOOL;
	bCollisionError									: BOOL;
	bCollision1Error								: BOOL;
	bCollision2Error								: BOOL;
	rtCollisionError								: R_TRIG;
	tonCollisionError								: TON;
	bCapBlow1										: BOOL;
	bCapBlow2										: BOOL;
	bCapBlow3										: BOOL;
	bCapBlow4										: BOOL;
	bPlaceDone										: BOOL;
	bTestCatch										: BOOL;
	iDisablingCase									: INT;
	bAdditionalBlow									: BOOL;
	bAxisYInPosition								: BOOL;
	bAxisZInPosition								: BOOL;
	bAxisZInPosition1								: BOOL;
	bAxisZInPosition2								: BOOL;
	bHomingWithoutJiesang							: BOOL;
	bCapLost										: ARRAY [1..4] OF BOOL;
	bAnyCapLost										: BOOL;

	trStepButton: R_TRIG;
	diManualModeCase								: DINT;
	bAxisYInHomePos									: BOOL;
	bAxisZInHomePos									: BOOL;
	bAxisZInTopPos									: BOOL;
	bAxisStrawCatcherHomePos						: BOOL;
	bCartesianInHomePos								: BOOL;										//Kartezjan znajduje sie na poz. home
	bCartesianInTopPos								: BOOL;
	bCartesianReady									: BOOL;										//Kartezjan gotowy do sekwencji
	rtCheckVacuumPart4								: R_TRIG;	


	FB_AxisY_ADS_Read								: FB_EcCoESdoRead;
	uiAxisY_ADS_Read								: UINT;
	tonAxisY_ADS_Read							    : TON;
	
	stAxisY_ADS										: ST_ADS_Read_Write;
	iAxisY_ADS_ReadCase								: INT;
	
	ftAxisY_ADS_Read								: F_TRIG;
	
	ftAxisY_ADS_Write								: F_TRIG;
	
	bSetPosition									: BOOL;
	FB_AxisY_ADS_Write								: FB_EcCoESdoWrite;
	tonAxisYLagDetction								: TON;		
	bCartesianInReadyPos							: BOOL;
	lrPreScrewerAxisSavedPosition					: LREAL;
	lrAxisZSavedPosition							: LREAL;
	
	bChangeSpeedRightLeft							: BOOL;
	rtPendantRightLeftFast							: R_TRIG;
	ftPendantRightLeftFast							: F_TRIG;
	bChangeSpeedUpDown								: BOOL;
	rtPendantUpDownFast								: R_TRIG;
	ftPendantUpDownFast								: F_TRIG;
	
	bAnyCapPresence									: BOOL;		//Obecna przynajmniej jedna nasadka
	tonWaitInPlacePos								: TON;
	diPreSCrewerHomePos								: DINT;

	//Synchronizacja osi podczas prowadzenia slomki
	fbGearInAxisZ									: MC_GearInDyn;
	fbGearInAxisZ_Screwer							: MC_GearIn;	
	fbGearInCatcherAxis								: MC_GearInDyn;
	fbGearOutAxisZ									: MC_GearOut;
	fbGearOutCatcherAxis							: MC_GearOut;
	fbVirtualAxis									: FB_AxisAX8000;
	fbGearInPos										: MC_GearInPos; 
	VirtualEna										: BOOL := TRUE;
	
	fbCamTableSelectAxisZ							: MC_CamTableSelect;
	fbCamInAxisZ									: MC_CamIn;
	fbCamOutAxisZ									: MC_CamOut;
	fbCamTableSelectCatcher							: MC_CamTableSelect;
	fbCamInAxisCatcher								: MC_CamIn;
	fbCamOutAxisCatcher								: MC_CamOut;	
	
	stCamTableIdAxisZ								: MC_CAM_ID;
	stCamTableAxisZRef								: MC_CAM_REF;
	arrTableAxisZ									: ARRAY[0..2, 0..1] OF LREAL;
	stCamTableIdCatcher								: MC_CAM_ID;
	stCamTableCatcherRef							: MC_CAM_REF;
	arrTableCatcher									: ARRAY[0..2, 0..1] OF LREAL;
	
	nAxisYSafetyState			AT%I*				: BYTE;	//Satatus safety 
	nAxisZSafetyState			AT%I*				: BYTE;	//Satatus safety 
	nAxisScrewSafetyState		AT%I*				: BYTE;	//Satatus safety 
	nAxisCatcherSafetyState		AT%I*				: BYTE;	//Satatus safety 
	
	uiAxisYTorqueLimit			AT%Q*				: UINT;
	
	rtChoseRecipe									: R_TRIG;
	tonCapCatcher1Open								: TON;
	bVirtualMove									: BOOL;		//Absolutny ruch  wirtualnej osi
	rtMove											: R_TRIG;
	ftMove											: F_TRIG;
	bVirtualAxisMove1								: BOOL;		//Ruch 1 wirtualnej osi
	bVirtualAxisMove2								: BOOL;		//Ruch 2 wirtualnej osi
	
	nMoveId											: INT;		//
	stVirtualMove_Out								: Tc2_MC2.ST_McOutputs;
	stVirtualMove1_Out								: Tc2_MC2.ST_McOutputs;	//struktura wyjsciowa ruchu wirtualnej osi
	stVirtualMove2_Out								: Tc2_MC2.ST_McOutputs; //struktura wyjsciowa ruchu wirtualnej osi
	bEnableLift										: BOOL	:= TRUE;
	bStrawCatcherLiftInHomePos						: BOOL;
	bMover1InPickPos								: BOOL; 			//nakrętka pobrana z wózka nr1
	bCapScrewed										: BOOL;				// nakrętka zakręcona
	rtSetEncoderOffsetAxisZ							: R_TRIG;
	tonStrawCatcherLiftInHomePos					: TON;				//łapacz słomek jest na poz bazowej
//	lrCatcherOffsetRegardingAxisZ					: LREAL;			//różnica położenia łapacza słomek odnośnie osi Z		
	bAlarmInit										: BOOL := TRUE;
	arrFbAllarm										: ARRAY [0..29] OF FB_TcAlarm;
	fbSourceInfo 									: FB_TcSourceInfo;
	sAxisAlarm										: STRING;	
	iSimulationCase									: INT;		
	bStrawCatcherLiftEnable							: BOOL;
	bReject											: BOOL;			//Odrzut aktywowany
	bTubeReject										: BOOL;			//Odrzut poprzez brak słomki
	iRejectCase										: INT;			
	lrAxisZ_RejectOffset							: LREAL;		//Offset odrzutu
	bAllSlotsVacuumStatus							: BOOL;			//Status wszsystkich aktywowanych ssawek
	arrVacuumStatus									: ARRAY [1..4] OF BOOL;	//status pojedynczych gniazd
	rtAxisZMoving									: R_TRIG;
	
	bTestCamCalculation								: BOOL;
END_VAR

IF bAlarmInit THEN
	ACT_ErrorInit();
END_IF


GVL_VIS.lrCapSorterPreScrewerStrawCatcherCVShow 			:= CatcherAxisRef.NcToPlc.ActPos;
GVL_VIS.lrCapSorterPreScrewerYAxisCVShow					:= CartesianYAxisRef.NcToPlc.ActPos;
GVL_VIS.lrCapSorterPreScrewerZAxisCVShow					:= CartesianZAxisRef.NcToPlc.ActPos;
GVL_VIS.lrCapSorterPreScrewerCAxisCVShow					:= PreScrewerAxisRef.NcToPlc.ActPos;

Signals();
ADS_Control();
Control();
ErrorHandling();
FBs();
CollisionAvoidance();


IF VirtualEna THEN
	ACT_VirtualAxisControl();
ELSE
	IF fbVirtualAxis.bEnable THEN
		fbVirtualAxis.Disable();
	END_IF	
END_IF

IF bTestCamCalculation THEN
	CamCalculation();
END_IF

ACTION ACT_ErrorInit:
bAlarmInit			:= FALSE;
fbSourceInfo.Clear();
fbSourceInfo.sName	:= wsLiteral_TO_UTF8(wsStationName);
fbSourceInfo.nId	:= iStationIndex;

arrFbAllarm[0].CreateEx(stEventEntry := TC_EVENTS.AlarmClass.CapPreScrewer_1130	, bWithConfirmation := FALSE, ipSourceInfo := fbSourceInfo);
arrFbAllarm[1].CreateEx(stEventEntry := TC_EVENTS.AlarmClass.CapPreScrewer_1131, bWithConfirmation := FALSE, ipSourceInfo := fbSourceInfo);
arrFbAllarm[2].CreateEx(stEventEntry := TC_EVENTS.AlarmClass.CapPreScrewer_1132, bWithConfirmation := FALSE, ipSourceInfo := fbSourceInfo);
arrFbAllarm[3].CreateEx(stEventEntry := TC_EVENTS.AlarmClass.CapPreScrewer_1133, bWithConfirmation := FALSE, ipSourceInfo := fbSourceInfo);
arrFbAllarm[4].CreateEx(stEventEntry := TC_EVENTS.AlarmClass.CapPreScrewer_1134, bWithConfirmation := FALSE, ipSourceInfo := fbSourceInfo);
arrFbAllarm[5].CreateEx(stEventEntry := TC_EVENTS.AlarmClass.CapPreScrewer_1135, bWithConfirmation := FALSE, ipSourceInfo := fbSourceInfo);
arrFbAllarm[6].CreateEx(stEventEntry := TC_EVENTS.AlarmClass.CapPreScrewer_1136, bWithConfirmation := FALSE, ipSourceInfo := fbSourceInfo);
arrFbAllarm[7].CreateEx(stEventEntry := TC_EVENTS.AlarmClass.CapPreScrewer_1137, bWithConfirmation := FALSE, ipSourceInfo := fbSourceInfo);
arrFbAllarm[8].CreateEx(stEventEntry := TC_EVENTS.AlarmClass.CapPreScrewer_1138, bWithConfirmation := FALSE, ipSourceInfo := fbSourceInfo);
arrFbAllarm[9].CreateEx(stEventEntry := TC_EVENTS.AlarmClass.CapPreScrewer_1139, bWithConfirmation := FALSE, ipSourceInfo := fbSourceInfo);
arrFbAllarm[10].CreateEx(stEventEntry := TC_EVENTS.AlarmClass.CapPreScrewer_1140, bWithConfirmation := FALSE, ipSourceInfo := fbSourceInfo);
arrFbAllarm[11].CreateEx(stEventEntry := TC_EVENTS.AlarmClass.CapPreScrewer_1141, bWithConfirmation := FALSE, ipSourceInfo := fbSourceInfo);
arrFbAllarm[12].CreateEx(stEventEntry := TC_EVENTS.AlarmClass.CapPreScrewer_1142, bWithConfirmation := FALSE, ipSourceInfo := fbSourceInfo);
arrFbAllarm[13].CreateEx(stEventEntry := TC_EVENTS.AlarmClass.CapPreScrewer_1143, bWithConfirmation := FALSE, ipSourceInfo := fbSourceInfo);
arrFbAllarm[14].CreateEx(stEventEntry := TC_EVENTS.AlarmClass.CapPreScrewer_1144, bWithConfirmation := FALSE, ipSourceInfo := fbSourceInfo);
arrFbAllarm[15].CreateEx(stEventEntry := TC_EVENTS.AlarmClass.CapPreScrewer_1145, bWithConfirmation := FALSE, ipSourceInfo := fbSourceInfo);
arrFbAllarm[16].CreateEx(stEventEntry := TC_EVENTS.AlarmClass.CapPreScrewer_1146, bWithConfirmation := FALSE, ipSourceInfo := fbSourceInfo);
arrFbAllarm[17].CreateEx(stEventEntry := TC_EVENTS.AlarmClass.CapPreScrewer_1147, bWithConfirmation := FALSE, ipSourceInfo := fbSourceInfo);
arrFbAllarm[18].CreateEx(stEventEntry := TC_EVENTS.AlarmClass.CapPreScrewer_1148, bWithConfirmation := FALSE, ipSourceInfo := fbSourceInfo);
arrFbAllarm[19].CreateEx(stEventEntry := TC_EVENTS.AlarmClass.CapPreScrewer_1149, bWithConfirmation := FALSE, ipSourceInfo := fbSourceInfo);
arrFbAllarm[20].CreateEx(stEventEntry := TC_EVENTS.AlarmClass.CapPreScrewer_1150, bWithConfirmation := FALSE, ipSourceInfo := fbSourceInfo);
arrFbAllarm[21].CreateEx(stEventEntry := TC_EVENTS.AlarmClass.CapPreScrewer_1151, bWithConfirmation := FALSE, ipSourceInfo := fbSourceInfo);
arrFbAllarm[22].CreateEx(stEventEntry := TC_EVENTS.AlarmClass.CapPreScrewer_1152, bWithConfirmation := FALSE, ipSourceInfo := fbSourceInfo);
arrFbAllarm[23].CreateEx(stEventEntry := TC_EVENTS.AlarmClass.CapPreScrewer_1153, bWithConfirmation := FALSE, ipSourceInfo := fbSourceInfo);
arrFbAllarm[24].CreateEx(stEventEntry := TC_EVENTS.AlarmClass.CapPreScrewer_1154, bWithConfirmation := FALSE, ipSourceInfo := fbSourceInfo);
arrFbAllarm[25].CreateEx(stEventEntry := TC_EVENTS.AlarmClass.CapPreScrewer_1155, bWithConfirmation := FALSE, ipSourceInfo := fbSourceInfo);
arrFbAllarm[26].CreateEx(stEventEntry := TC_EVENTS.AlarmClass.CapPreScrewer_1156, bWithConfirmation := FALSE, ipSourceInfo := fbSourceInfo);
arrFbAllarm[27].CreateEx(stEventEntry := TC_EVENTS.AlarmClass.CapPreScrewer_1157, bWithConfirmation := FALSE, ipSourceInfo := fbSourceInfo);
arrFbAllarm[28].CreateEx(stEventEntry := TC_EVENTS.AlarmClass.CapPreScrewer_1158, bWithConfirmation := FALSE, ipSourceInfo := fbSourceInfo);
arrFbAllarm[29].CreateEx(stEventEntry := TC_EVENTS.AlarmClass.CapPreScrewer_1159, bWithConfirmation := FALSE, ipSourceInfo := fbSourceInfo);
END_ACTION

ACTION ACT_VirtualAxisControl:
IF fbVirtualAxis.bDisabled THEN
	fbVirtualAxis.bEnable	:= TRUE;
	fbVirtualAxis.Power();
END_IF


rtMove(CLK := bVirtualMove);
ftMove(CLK := bVirtualMove);

IF rtMove.Q THEN
	bVirtualAxisMove2 							S= stVirtualMove1_Out.Busy; 
	bVirtualAxisMove1 							S= NOT bVirtualAxisMove2;
ELSIF ftMove.Q THEN
	bVirtualAxisMove1							R= TRUE;	
    bVirtualAxisMove2							R= TRUE;	
END_IF


IF NOT stVirtualMove2_Out.Busy AND NOT stVirtualMove2_Out.Done THEN
	nMoveId					:= 1;
	stVirtualMove_Out		:= stVirtualMove1_Out ;
ELSE
	nMoveId					:= 2;
	stVirtualMove_Out		:= stVirtualMove2_Out;
END_IF

stVirtualMove1_Out 			:= fbVirtualAxis.MoveAbsolute(bExecute := bVirtualAxisMove1);
stVirtualMove2_Out 			:= fbVirtualAxis.MoveAbsolute2(bExecute := bVirtualAxisMove2);


fbVirtualAxis.fAcceleration;//						:= stParameters.lrPickerAcceleration;	//100_000_000.0;
fbVirtualAxis.fDeceleration;//						:= stParameters.lrPickerAcceleration;	//100_000_000.0;
fbVirtualAxis.fJerk;//							:= stParameters.lrPickerJerk;// 	1_000_000;//100_000_000_000;  








fbGearInPos.SyncMode.GearInSyncMode							:= E_GearInSyncMode.GEARINSYNCMODE_POSITIONBASED;	//Synchronizacja według pozycji mastera
fbGearInPos.SyncMode.GearInSync_OpMask_DetailedErrorCodes 	:= TRUE;	//szczególowy opis błedów
fbGearInPos.SyncMode.GearInSync_CheckMask_MaxVelo 			:= TRUE;	//vSlave | ≤ vSlaveMax
fbGearInPos.SyncMode.GearInSync_CheckMask_MaxAcc 			:= TRUE;	//accSlave ≤ accSlaveMax
fbGearInPos.SyncMode.GearInSync_CheckMask_MaxDec 			:= TRUE;	//decSlave ≤ decSlaveMax
fbGearInPos.SyncMode.GearInSync_CheckMask_MaxJerk 			:= TRUE;	//jSlave ≤ jSlaveMax
fbGearInPos.SyncMode.GearInSync_CheckMask_MinPos			:= TRUE;
fbGearInPos.SyncMode.GearInSync_CheckMask_MaxPos			:= TRUE;
fbGearInPos.Options.PositionLimitMax;//						:= 450.0;//SEL(stParameters.lrCartesianCatchZPosition>450, stParameters.lrCartesianCatchZPosition, 450);
fbGearInPos.Options.PositionLimitMin						:= 0.0;
END_ACTION

ACTION ADS_Control:
tonAxisY_ADS_Read(PT := T#250MS);

(*	//Wyłączenie krańcówek podczas bazowania na zderzak wózek 1
			IF eState = E_Station.eHoming AND bAdvancedHoming AND uiMover1ADS_Read <> 0 THEN	//	ADS_Read = 0 - no limit switch
				uiMover1ADS_Write				:= 0;                                           //			 = 1 - NC
				FB_Mover1ADS_Write.bExecute		:= TRUE;                                        //			 = 2 - NO
			ELSIF eState <> E_Station.eHoming AND uiMover1ADS_Read <> 1 THEN	                
				uiMover1ADS_Write				:= 1;                                           
				FB_Mover1ADS_Write.bExecute		:= TRUE;                                        
			END_IF
		
			ftMover1ADS_Write(CLK := FB_Mover1ADS_Write.bBusy);
			FB_Mover1ADS_Write.bExecute			R= ftMover1ADS_Write.Q;
			
		
	//Wyłączenie krańcówek podczas bazowania na zderzak wózek 2
			IF eState = E_Station.eHoming AND bAdvancedHoming AND uiMover2ADS_Read <> 0 THEN
				uiMover2ADS_Write				:= 0;
				FB_Mover2ADS_Write.bExecute		:= TRUE;
			ELSIF eState <> E_Station.eHoming AND uiMover2ADS_Read <> 1 THEN	 
				uiMover2ADS_Write				:= 1;
				FB_Mover2ADS_Write.bExecute		:= TRUE;
			END_IF
		\
			ftMover2ADS_Write(CLK := FB_Mover2ADS_Write.bBusy);
			FB_Mover2ADS_Write.bExecute			R= ftMover2ADS_Write.Q;
		
		
	//odswieżanie parametrów krańcówek hardwerowych wózek 1
			ftMover1ADS_Read(CLK := FB_Mover1ADS_Read.bBusy);
			FB_Mover1ADS_Read.bExecute			S= (tonAxisY_ADS_Read.Q AND NOT ftMover1ADS_Read.Q);
			FB_Mover1ADS_Read.bExecute			R= ftMover1ADS_Read.Q;
			
			tonAxisY_ADS_Read.IN				:= NOT tonAxisY_ADS_Read.Q;
	
	//odswieżanie parametrów krańcówek hardwerowych wózek 2
			ftMover2ADS_Read(CLK := FB_Mover2ADS_Read.bBusy);
			FB_Mover2ADS_Read.bExecute			S= (tonAxisZ_ADS_Read.Q AND NOT ftMover2ADS_Read.Q);
			FB_Mover2ADS_Read.bExecute			R= ftMover2ADS_Read.Q;
			
			tonAxisZ_ADS_Read.IN				:= NOT tonAxisZ_ADS_Read.Q;*)

////////////////////////////////////////////////////////////////////////////////////////////////////////////////

//CASE iAxisY_ADS_ReadCase OF
//	
//	0://Odczyt momentu
//	FB_AxisY_ADS_Read.nSubIndex				:= 16#0;
//	FB_AxisY_ADS_Read.nIndex				:= 16#60E0;
//	                                		
//	stAxisY_ADS.stSts.uiTorq				:= uiAxisY_ADS_Read;
//	                                		
//		IF ftAxisY_ADS_Read.Q THEN  		
//			iAxisY_ADS_ReadCase				:= 1;
//		END_IF
//	
//	1://Odczyt krancowek

//	
//END_CASE

		//Wyłączenie krańcówek podczas bazowania na zderzak oś Y
	IF eState = E_Station.eHoming AND bAdvancedHoming AND stAxisY_ADS.uiHardwerLimitSwitch <> 0 THEN//	ADS_Read = 0 - no limit switch
		FB_AxisY_ADS_Write.nSubIndex			:= 16#1;											//			 = 1 - NC
		FB_AxisY_ADS_Write.nIndex				:= 16#3003;                                         //			 = 2 - NO
		stAxisY_ADS.stCtr.siHardwerLimitSwitch	:= 0;                   
		FB_AxisY_ADS_Write.bExecute				:= TRUE;                
	ELSIF eState <> E_Station.eHoming AND stAxisY_ADS.uiHardwerLimitSwitch <> 1 THEN	
		FB_AxisY_ADS_Write.nSubIndex			:= 16#1;	
        FB_AxisY_ADS_Write.nIndex				:= 16#3003;
        stAxisY_ADS.stCtr.siHardwerLimitSwitch	:= 1;      
        FB_AxisY_ADS_Write.bExecute				:= TRUE;                                    
	END_IF
	
	ftAxisY_ADS_Write(CLK := FB_AxisY_ADS_Write.bBusy);
	FB_AxisY_ADS_Write.bExecute			R= ftAxisY_ADS_Write.Q;
	
	

	//odswieżanie parametrów krańcówek hardwerowych oś Y
	FB_AxisY_ADS_Read.nSubIndex					:= 16#1;
	FB_AxisY_ADS_Read.nIndex					:= 16#3003;
	
	ftAxisY_ADS_Read(CLK := FB_AxisY_ADS_Read.bBusy);
	FB_AxisY_ADS_Read.bExecute					S= (tonAxisY_ADS_Read.Q AND NOT ftAxisY_ADS_Read.Q);
	FB_AxisY_ADS_Read.bExecute					R= ftAxisY_ADS_Read.Q;
	stAxisY_ADS.uiHardwerLimitSwitch			:= uiAxisY_ADS_Read;
	
	tonAxisY_ADS_Read.IN						:= NOT tonAxisY_ADS_Read.Q;
	
	IF NOT bAdvancedHoming AND (stAxisY_ADS.stCtr.uiNegativeTorqueLimit <> 2000 OR stAxisY_ADS.stCtr.uiPositiveTorqueLimit <> 2000 OR uiAxisYTorqueLimit <> 2000) THEN	
		stAxisY_ADS.stCtr.uiNegativeTorqueLimit			:= 2000;	
		stAxisY_ADS.stCtr.uiPositiveTorqueLimit			:= 2000;
		uiAxisYTorqueLimit								:= 2000;
	END_IF
END_ACTION

ACTION CamCalculation:

//Tablica punktów dla osi prowadzenia słomki:
		//Pozycję Mastera:
	arrTableCatcher[0,0]			:= 0.0;		//Początek ruchu 
	arrTableCatcher[1,0]			:= (stParameters.lrCatcherCatchingPosition  - (stParameters.lrBottleHight - stParameters.lrCatcherHightSV - 40));	//Punkt nad butelką 40mm ---> 40mm grubość chwytaków /////
	//Sprawdzanie czy nie przekraczamy dolny limit (min 2mm)
	arrTableCatcher[1,0]			:= SEL((stParameters.lrCatcherCatchingPosition - arrTableCatcher[1,0] < 2.0), arrTableCatcher[1,0], (stParameters.lrCatcherCatchingPosition - 2.0));
	arrTableCatcher[2,0]			:= 1000.0;	//Koniec dojazdu mastera
	                        		
		//Pozycję Slave:    		
	arrTableCatcher[0,1]			:= 0.0;	//Początek ruchu 
	arrTableCatcher[1,1]			:= arrTableCatcher[1,0];	//Punkt nad butelką
	arrTableCatcher[2,1]			:= arrTableCatcher[1,0];	//Koniec dojazdu mastera

//Tablica punktów dla osi Z:
		//Pozycję Mastera:
	arrTableAxisZ[0,0]				:= 0.0;	//Początek ruchu 
	arrTableAxisZ[1,0]				:= (stParameters.lrCapHight - GVL_Recipe.lrCapSorterCapNeckHightShow - GVL_Recipe.lrCapSorterPreScrewerCheckValveShow - 30.0);	//Punkt Synchronizacji (~10mm od końca słomki)
	arrTableAxisZ[2,0]				:= 1000.0;	//Koniec dojazdu mastera
		//Pozycję Slave:    		
	arrTableAxisZ[0,1]				:= 0.0;	//Początek ruchu 
	arrTableAxisZ[1,1]				:= 0.0;	//Punkt Synchronizacji (~10mm od końca słomki)
	arrTableAxisZ[2,1]				:= 1000.0 - arrTableAxisZ[1,0];	//Koniec dojazdu mastera

//stCamTableCatcherRef.pArray			:= ADR(arrTableCatcher);
//stCamTableCatcherRef.ArraySize		:= SIZEOF(arrTableCatcher);
//stCamTableCatcherRef.TableType		:= MC_TableType.MC_TABLETYPE_NONEQUIDISTANT;
//stCamTableCatcherRef.NoOfRows		:= 3;
//stCamTableCatcherRef.NoOfColumns 	:= 2;
//stCamTableIdCatcher					:= SEL(stCamTableIdCatcher=0, stCamTableIdCatcher, 1);
//
//stCamTableAxisZRef.pArray			:= ADR(arrTableAxisZ);
//stCamTableAxisZRef.ArraySize		:= SIZEOF(arrTableAxisZ);
//stCamTableAxisZRef.TableType		:= MC_TableType.MC_TABLETYPE_NONEQUIDISTANT;
//stCamTableAxisZRef.NoOfRows			:= 3;
//stCamTableAxisZRef.NoOfColumns 		:= 2;
//stCamTableIdAxisZ					:= SEL(stCamTableIdAxisZ=0, stCamTableIdAxisZ, 2);
END_ACTION

ACTION CollisionAvoidance:

//bCollision1Error			:= 	mcCartesianYPower.Override = 0;
//bCollision2Error			:= 	mcCartesianZPower.Override = 0 OR mcCartesianZStop.Execute = TRUE;

tonCollisionError(IN := bCollision1Error OR bCollision1Error, PT := T#3S);
rtCollisionError(CLK := tonCollisionError.Q);

bCollisionWithMoverArea := CartesianZAxisRef.NcToPlc.ActPos < 354.0 AND CartesianYAxisRef.NcToPlc.ActPos < 65.0;

IF CartesianZAxisRef.NcToPlc.ActPos < 206 AND NOT bSetPosition THEN	
	
	IF CartesianYAxisRef.NcToPlc.SetPos <= 354 AND NOT CartesianYAxisRef.Status.PositiveDirection THEN
		mcCartesianYPower.Override 	:= 0;
//		bHomingDone					:= FALSE;
//	ELSIF CartesianYAxisRef.NcToPlc.SetPos >= 111 AND NOT CartesianYAxisRef.Status.NegativeDirection THEN
//		mcCartesianYPower.Override 	:= 0;
	ELSIF CartesianYAxisRef.Status.PositiveDirection THEN
		mcCartesianYPower.Override 	:= 100;	
	END_IF	
	
ELSE
	mcCartesianYPower.Override := 100;	
END_IF


//IF CartesianYAxisRef.NcToPlc.ActPos < 160 AND CartesianZAxisRef.NcToPlc.SetPos < 358 
//	OR CartesianYAxisRef.NcToPlc.ActPos > 200 AND CartesianZAxisRef.NcToPlc.SetPos < 185 THEN
//	
//		IF CartesianZAxisRef.Status.NegativeDirection AND CartesianZAxisRef.Status.Moving THEN
//			mcCartesianZStop.Execute						:= TRUE;
//			mcCartesianZMoveAbsolute.Execute				:= FALSE;
//			mcCartesianZMoveAbsolute2.Execute				:= FALSE;
//			
//			bHomingDone					:= FALSE;
//		ELSE
//			mcCartesianZStop.Execute						:= FALSE;
//		END_IF
//END_IF


//IF CartesianYAxisRef.NcToPlc.ActPos > 200 AND CartesianZAxisRef.NcToPlc.ActPos - CatcherAxisRef.NcToPlc.ActPos < 200 THEN
//	mcCartesianZPower.Override :=F_Scaling_Limit(
//									In:=ABS(CartesianZAxisRef.NcToPlc.ActPos - CatcherAxisRef.NcToPlc.ActPos),
//									INMin:=0, INMax:= 200, OUTMin:=0, OUTMax:=100);
//ELSE
//	mcCartesianZPower.Override	:= 100;
//END_IF



CartesianZAxisRef.NcToPlc.ActPos;
CartesianZAxisRef.PlcToNc.ExtSetPos;

CartesianYAxisRef.NcToPlc.ActPos;
CartesianYAxisRef.PlcToNc.ExtSetPos;
END_ACTION

ACTION Control:
	(** TIMERY**)
//	tonGripper1ReliseDelay	(IN:=	NOT bGripper1Actuator, 					PT:=T#50MS);	//bylo 80
//	tonGripper2ReliseDelay	(IN:=	NOT bGripper2Actuator, 					PT:=T#50MS);	//bylo 80
                                 	
//	tonGripper1Delay		(IN:=	bGripper1Actuator OR iTool = 2, 						PT:=T#150MS);	//bylo 200  /// jednak 150
//	tonGripper2Delay		(IN:=	bGripper2Actuator OR iTool = 2, 						PT:=T#150MS);	//bylo 200 /// a jednak 150
                            																																								// Nie moze być 60 bo nalicza 60 i powyzej 360 sie przekręca																			
//	tonTightScrewing1Timer	(IN:=	(eRunningState=E_GripperScrewer.eScrewing) AND NOT tonTightScrewing1Timer.Q AND mcScrewer1MoveVelocity.Execute AND mcScrewer1MoveVelocity.InVelocity AND Screwing1AxisRef.NcToPlc.ActVelo < 100 (*AND ABS(Screwing1AxisRef.NcToPlc.PosDiff)>60 *) AND NOT bScrewed1,PT:=INT_TO_TIME(iScrewTightTime));
//	tonTightScrewing2Timer	(IN:=	(eRunningState=E_GripperScrewer.eScrewing) AND NOT tonTightScrewing2Timer.Q AND mcScrewer2MoveVelocity.Execute AND mcScrewer2MoveVelocity.InVelocity AND Screwing2AxisRef.NcToPlc.ActVelo < 100 (*AND ABS(Screwing2AxisRef.NcToPlc.PosDiff)>60 *) AND NOT bScrewed2,PT:=INT_TO_TIME(iScrewTightTime));

//	tonTightScrewing1TimerAndOpenedGripper(IN:=bScrewed1,	PT:=T#100MS);
//	tonTightScrewing2TimerAndOpenedGripper(IN:=bScrewed2,	PT:=T#100MS);	
	
//	tonMomentaryScrewing1Timer	(IN:=	(eRunningState=E_GripperScrewer.eScrewing)	AND NOT tonMomentaryScrewing1Timer.Q AND 
//											mcScrewer1TorqueControl.Execute 		AND 
//											Screwing1AxisRef.NcToPlc.ActVelo < 100  AND NOT bScrewed1,
//										PT:=INT_TO_TIME(iScrewTightTime));
//	tonMomentaryScrewing2Timer	(IN:=	(eRunningState=E_GripperScrewer.eScrewing)	AND NOT tonMomentaryScrewing2Timer.Q AND 
//											mcScrewer2TorqueControl.Execute 		AND 
//											Screwing2AxisRef.NcToPlc.ActVelo < 100  AND NOT bScrewed2,
//										PT:=INT_TO_TIME(iScrewTightTime));
	
//	tonHoldingTimer			(IN:=	(eRunningState=E_GripperScrewer.eHolding ),	PT:=INT_TO_TIME(iScrewTightTime));
                  	
	tonDelayServoOn			(IN:=	(eState = E_Station.ePreparingToReady), PT:=T#20S); //bylo 1,2s
	tonResetting			(IN:=	(eState = E_Station.eResetting), 		PT:=T#4S);
	
	rtResetCommands			(CLK:=	eState = E_Station.eReady (* OR *)		,Q=>); //Triger do resetu zmienych
//	tonDelayBeforeResetLag 	(IN:=	iPreparingToReadyCase=10, 				PT:=T#10MS);

//tonFindingScrewDelay 	(IN:=	iFindingScrewCASE = 50, 				PT:=T#0MS);
//	tonStoppingCaseError	(IN:=	eState = E_Station.eStopping AND  (iStoppingCase = 30 OR iStoppingCase = 40), PT:=T#10S); 
	
	
	(*****Wyłączenie enable*****)
	IF NOT bEnable AND NOT bError THEN
		IF eState <> E_Station.eDisabled AND eState <> E_Station.ePreparingToDisable AND eState <> E_Station.eAborting AND  eState <> E_Station.eAborted THEN
			eState 				:= E_Station.ePreparingToDisable; 
		END_IF	
	END_IF

	IF eState <> E_Station.eManualMovement THEN
		
		bManualCapCatcher1								:= FALSE;
		bManualCapCatcher2								:= FALSE;
		bManualCapCatcher3								:= FALSE;
		bManualCapCatcher4					    		:= FALSE;
		bManualCapSucker1								:= FALSE;
		bManualCapSucker2								:= FALSE;
		bManualCapSucker3								:= FALSE;
		bManualCapSucker4								:= FALSE;

	END_IF


	(*****Estop*****)
	IF NOT bEstop  THEN	
		IF eState <> E_Station.eAborted AND eState <> E_Station.eAborting AND eState <> E_Station.eDisabled THEN
				iAbortingCASE		:=	0;
				eState 				:=	E_Station.eAborting; 
				
				//Jeżeli cartezjan nie jest na pozycji Ready --> wymus bazowanie
				//IF eRunningState <> E_CapPreScrewer.eReady THEN
				//	bHomingDone				:= FALSE;
				//	bHomingWithoutJiesang	:= fbBottleCatch1Station.bHomingDone;
				//END_IF
				
		END_IF
	END_IF
	
	IF NOT bRun AND bMissingCaps THEN
		bCycleNotDone				:= FALSE;
		bMissingCaps				:= FALSE;
	END_IF

	
	CASE eState OF
	/////////////////////////////	
		E_Station.eDisabled: 					// Stan nieaktywnosci (Stacja wyłączona) 
			bHomingDone				:= FALSE;
			bHomingWithoutJiesang	:= FALSE;
		
			IF bEnable  THEN
				eState 				:= E_Station.ePreparingToReady; 
			END_IF 
			
    /////////////////////////////	    
		E_Station.eAborted: 					// Stan bezpiecznego zatrzymania (po Abortingu) 
			fbGearOutAxisZ.Execute				:= CartesianZAxisRef.Status.Coupled;
			fbGearOutCatcherAxis.Execute		:= CatcherAxisRef.Status.Coupled;
		

			IF bEStop THEN
		//		bHomingDone			R= (eRunningState <> E_CapPreScrewer.eReady);
				eState 				:= E_Station.ePreparingToReady;
			END_IF
			
	/////////////////////////////	
		E_Station.eAborting:                 	// Stan bezpiecznego zatrzymywania (po EStopie)
		
			CASE iAbortingCASE OF   
				0: //Czyszczenie
					ResetCommands(); 
					iAbortingCASE	:=	iAbortingCASE	+	10;
//					iCountAborting	:=	iCountAborting	+	1;
				10: //Stop
					mcCartesianYPower.Override		:=	100;
					mcCartesianZPower.Override		:=	100;
					mcPreScrewerPower.Override		:=	100;
					mcCatcherPower.Override			:=	100;

		
					//F NOT mcHeightStop.Error AND NOT mcScrewer1Stop.Error AND NOT mcScrewer2Stop.Error THEN
					mcCartesianYStop.Execute		:=	TRUE;
					mcCartesianZStop.Execute		:=	TRUE;
					mcPreScrewerStop.Execute		:=	TRUE;
					mcCatcherStop.Execute			:= TRUE;

					iAbortingCASE					:=	iAbortingCASE	+	10;	
					//ELSE
				(*	mcHeightStop.Execute			:=	FALSE;
					mcScrewer1Stop.Execute			:=	FALSE;
					mcScrewer2Stop.Execute			:=	FALSE;
					bHeightServoPower				:=	FALSE;
					bScrewer1ServoPower				:=	FALSE;
					bScrewer2ServoPower				:=	FALSE;*)
					//END_IF	
					iCountAborting	:=	iCountAborting	+	1;						
				20: //Stop Done		
				
					IF 
						(mcCartesianYStop.Done  OR mcCartesianYStop.Error OR NOT bCartesianYServoPower) AND
						(mcCartesianZStop.Done  OR mcCartesianZStop.Error OR NOT bCartesianZServoPower) AND
						(mcCatcherStop.Done  OR mcCatcherStop.Error OR NOT bCatcherPower) AND
						(mcPreScrewerStop.Done  OR mcPreScrewerStop.Error OR NOT bPreScrewerPower)					
						 THEN
							bCartesianYServoPower		:=	FALSE;
							bCartesianZServoPower		:=	FALSE;	
							bCatcherPower				:=	FALSE;
							bPreScrewerPower			:=	FALSE;						
	
							iAbortingCASE			:=	iAbortingCASE	+	10;			
					END_IF	
					
				30: //Wyjście
					ResetCommands(); 
					eState							:=	E_Station.eAborted; 
			//		eRunningState					:=	E_CapPreScrewer.eReady;
			END_CASE
			
	/////////////////////////////			
		E_Station.eError:                 	 	// Stan błędu 	
		
			fbGearOutAxisZ.Execute				:= CartesianZAxisRef.Status.Coupled;
			mcCartesianZStop.Execute			:= CartesianZAxisRef.Status.Moving;
			
			fbGearOutCatcherAxis.Execute		:= CatcherAxisRef.Status.Coupled;
			mcCatcherStop.Execute				:= PreScrewerAxisRef.Status.Moving;


			IF bReset THEN
				eState 						:= E_Station.eResetting;
				iTestResetting					:= iTestResetting	+	1;			
			END_IF
			
	/////////////////////////////
		E_Station.eResetting:					// Stan resetowania bledu (po Errorze)
		
			diMover1VacuumRetry[1]				:= 0;
			diMover1VacuumRetry[2]				:= 0;
			diMover1VacuumRetry[3]				:= 0;
			diMover1VacuumRetry[4]				:= 0;
			fbVirtualAxis.Reset(bExecute := fbVirtualAxis.bError);	

			//Procedura obsługi resetu w zależności od błędu
			CASE udiErrorID OF
			
				//Error 2 - BŁĄD SERWA WÓZKA 1
				//Error 3 - BŁĄD SERWA WÓZKA 2			
				0, 1129..1132, 1151..1159:	

					CASE iErrorResseting2 OF
					0:
						IF mcCartesianYPower.Status THEN
							bCartesianYServoPower 	:= FALSE;
						END_IF
						
						IF mcCartesianZPower.Status THEN
							bCartesianZServoPower 	:= FALSE;
						END_IF

						IF mcCatcherPower.Status THEN
							bCatcherPower			:= FALSE;
						END_IF
						
						IF mcPreScrewerPower.Status THEN
							bPreScrewerPower 		:= FALSE;
						END_IF
		
						fbCartesianYHardReset		(Execute:=TRUE,	Axis:=CartesianYAxisRef);
						fbCartesianZHardReset		(Execute:=TRUE,	Axis:=CartesianZAxisRef);
						fbPreScrewerHardReset		(Execute:=TRUE,	Axis:=PreScrewerAxisRef);
						fbCatcherHardReset			(Execute:=TRUE,	Axis:=CatcherAxisRef);
						mcCartesianYSoftReset		(Execute:=TRUE,	Axis:=CartesianYAxisRef); 
						mcCartesianZSoftReset		(Execute:=TRUE,	Axis:=CartesianZAxisRef);
						mcPreScrewerSoftReset		(Execute:=TRUE,	Axis:=PreScrewerAxisRef);
						mcCatcherSoftReset			(Execute:=TRUE,	Axis:=CatcherAxisRef);
						fbVirtualAxis.Reset(bExecute := fbVirtualAxis.bError);						
		
						IF bEnable THEN
							bCartesianYServoPower 	:= TRUE;
							bCartesianzServoPower 	:= TRUE;
							bPreScrewerPower		:= TRUE;
							bCatcherPower			:= TRUE;	
						END_IF
						

						IF 
						( NOT fbCartesianYHardReset.Busy AND NOT mcCartesianYSoftReset.Busy AND (mcCartesianYPower.Status OR NOT bEnable) AND NOT CartesianYAxisRef.Status.Error ) AND
						( NOT fbCartesianZHardReset.Busy AND NOT mcCartesianZSoftReset.Busy AND (mcCartesianZPower.Status OR NOT bEnable) AND NOT CartesianZAxisRef.Status.Error ) AND
						( NOT fbPreScrewerHardReset.Busy AND NOT mcPreScrewerSoftReset.Busy AND (mcPreScrewerPower.Status OR NOT bEnable) AND NOT PreScrewerAxisRef.Status.Error ) AND
						( NOT fbCatcherHardReset.Busy AND NOT mcCatcherSoftReset.Busy AND (mcCatcherPower.Status OR NOT bEnable) AND NOT CatcherAxisRef.Status.Error AND (NOT fbVirtualAxis.bError OR NOT VirtualEna))
						
						THEN
							fbCartesianYHardReset		(Execute:=FALSE,	Axis:=CartesianYAxisRef);
							fbCartesianZHardReset		(Execute:=FALSE,	Axis:=CartesianZAxisRef);
							fbPreScrewerHardReset		(Execute:=FALSE,	Axis:=PreScrewerAxisRef);
							fbCatcherHardReset			(Execute:=FALSE,	Axis:=CatcherAxisRef);
							mcCartesianYSoftReset		(Execute:=FALSE,	Axis:=CartesianYAxisRef); 
							mcCartesianZSoftReset		(Execute:=FALSE,	Axis:=CartesianZAxisRef);
							mcPreScrewerSoftReset		(Execute:=FALSE,	Axis:=PreScrewerAxisRef);
							mcCatcherSoftReset			(Execute:=FALSE,	Axis:=CatcherAxisRef);		
							


							bError								:=	FALSE;
							iErrorResseting2					:=	0;	
							udiCartesianXServoErrorNr			:=	0;
							udiCartesianZServoErrorNr			:=	0;
							sErrorDescription					:=	'';
							sErrorDescription2					:=	'';

							udiErrorID							:=	0;
						END_IF	
					END_CASE
				
				1133..1141:
				//fbCartesianZHardReset(Execute:=CartesianZAxisRef.Status.Error,	Axis:=CartesianZAxisRef);
				//mcCartesianZSoftReset(Execute:=CartesianZAxisRef.Status.Error,	Axis:=CartesianZAxisRef);	
				//
				//IF (NOT CartesianZAxisRef.Status.Error AND NOT fbCartesianZHardReset.Busy
				//	AND NOT mcCartesianZSoftReset.Busy AND mcCartesianZPower.Status) THEN
				//		mcCartesianZMoveAbsolute.Execute		:= TRUE;		
				//		mcCartesianZMoveAbsolute.Position		:= 450.0;
				//		mcCartesianZMoveAbsolute.Acceleration	:= 1000.0;
				//		mcCartesianZMoveAbsolute.Deceleration	:= 1000.0;
				//		mcCartesianZMoveAbsolute.Velocity		:= 15.0;
				//END_IF	
				//
				//IF mcCartesianZMoveAbsolute.Done THEN
					bStrawCatcherActuatorIn						:= FALSE;
					bStrawCatcherActuatorOut					:= FALSE;
					mcCartesianZMoveAbsolute.Execute			:= FALSE;
					bError										:= FALSE;
					iErrorResseting2							:= 0;	
					udiCartesianXServoErrorNr					:= 0;
					udiCartesianZServoErrorNr					:= 0;
					sErrorDescription							:= '';
					sErrorDescription2							:= '';
                	                                    		   
					udiErrorID									:= 0;	
				//END_IF	
	
			
				//Error 6 - BŁAD POZYCJI MINIMALNEJ PODNOŚNIKA 
				6:
					IF NOT fbStrawCatcherLift.bError THEN
						bError										:= FALSE;						
					END_IF			
				1142..1150:
				
					diMover2VacuumRetry[1]				:= 0;
					diMover2VacuumRetry[2]				:= 0;
					diMover2VacuumRetry[3]				:= 0;
					diMover2VacuumRetry[4]				:= 0;
					bError								:=	FALSE;
					sErrorDescription					:=	'';
					sErrorDescription2					:=	'';
				ELSE
					bError								:=	FALSE;	
			END_CASE	
			
			IF NOT bError THEN
				udiErrorID 						:=	0;
   				sErrorDescription 				:=	'';                       			
				eState 							:=	E_Station.ePreparingToReady;
			ELSIF tonResetting.Q THEN     
				ResetCommands();       	
				eState 							:=	E_Station.eError;
			END_IF
        
	/////////////////////////////
		E_Station.eManualMovement:     			// Stan ruchów manualnych  
		
			IF bHoming THEN
				eState 				:= E_Station.eHoming; 
			END_IF
       
			ManualMovements(); 
			//Wyjście z trybu serwisowego
			IF NOT bManualMovement THEN
					//bManualGripper1				:=	FALSE;
					//bManualGripper2				:=	FALSE;		
	

			
					mcCartesianYPower.Override		:= 100;
					mcCartesianZPower.Override		:= 100;
					mcPreScrewerPower.Override		:= 100;
					mcCatcherPower.Override			:= 100;
//					IF
//						Height1AxisRef.NcToPlc.ActPos	<=	lrHeightReadyPosition OR
//						Height2AxisRef.NcToPlc.ActPos	<=	lrHeightReadyPosition
//					THEN
//						mcHeight1MoveAbsolute.Execute		:=	TRUE;
//						mcHeight1MoveAbsolute.Position		:=	lrHeightReadyPosition;
						
